LIN {X 0,Y 467.611,Z 154.239,A -85,B 0,C 180,E1 -7725.196,E2 -7725.196} C_VEL
LIN {X 0,Y 467.661,Z 154.233,A -85,B 0,C 180,E1 -7727.854,E2 -7727.854} C_VEL
LIN {X 0,Y 467.686,Z 154.231,A -85,B 0,C 180,E1 -7731.357,E2 -7731.357} C_VEL
LIN {X 0,Y 467.748,Z 154.222,A -85,B 0,C 180,E1 -7733.962,E2 -7733.962} C_VEL
LIN {X 0,Y 467.864,Z 154.208,A -85,B 0,C 180,E1 -7737.417,E2 -7737.417} C_VEL
LIN {X 0,Y 467.888,Z 154.205,A -85,B 0,C 180,E1 -7740,E2 -7740} C_VEL
LIN {X 0,Y 467.863,Z 154.208,A -85,B 0,C 180,E1 -7742.582,E2 -7742.582} C_VEL
LIN {X 0,Y 467.747,Z 154.225,A -85,B 0,C 180,E1 -7746.037,E2 -7746.037} C_VEL
LIN {X 0,Y 467.662,Z 154.235,A -85,B 0,C 180,E1 -7748.643,E2 -7748.643} C_VEL
LIN {X 0,Y 467.382,Z 154.273,A -85,B 0,C 180,E1 -7751.272,E2 -7751.272} C_VEL
LIN {X 0,Y 467.316,Z 155.866,A -85,B 0,C 180,E1 -7753.037,E2 -7753.037} C_VEL
LIN {X 0,Y 467.288,Z 158.633,A -85,B 0,C 180,E1 -7755.727,E2 -7755.727} C_VEL
LIN {X 0,Y 467.15,Z 161.596,A -85,B 0,C 180,E1 -7758.594,E2 -7758.594} C_VEL
LIN {X 0,Y 467.051,Z 165.325,A -85,B 0,C 180,E1 -7762.097,E2 -7762.097} C_VEL
LIN {X 0,Y 467.008,Z 168.875,A -85,B 0,C 180,E1 -7765.452,E2 -7765.452} C_VEL
LIN {X 0,Y 466.965,Z 172.431,A -85,B 0,C 180,E1 -7768.79,E2 -7768.79} C_VEL
LIN {X 0,Y 466.958,Z 173.469,A -85,B 0,C 180,E1 -7769.738,E2 -7769.738} C_VEL
LIN {X 0,Y 470.291,Z 187.316,A -85,B 0,C 180,E1 -7770.288,E2 -7770.288} C_VEL
LIN {X 0,Y 470.011,Z 200.111,A -85,B 0,C 180,E1 -7770.868,E2 -7770.868} C_VEL
LIN {X 0,Y 469.534,Z 212.003,A -85,B 0,C 180,E1 -7771.592,E2 -7771.592} C_VEL
LIN {X 0,Y 469.166,Z 222.158,A -85,B 0,C 180,E1 -7772.379,E2 -7772.379} C_VEL
LIN {X 0,Y 468.706,Z 232.669,A -85,B 0,C 180,E1 -7773.385,E2 -7773.385} C_VEL
LIN {X 0,Y 468.248,Z 242.269,A -85,B 0,C 180,E1 -7774.534,E2 -7774.534} C_VEL
LIN {X 0,Y 467.748,Z 251.276,A -85,B 0,C 180,E1 -7775.872,E2 -7775.872} C_VEL
LIN {X 0,Y 467.449,Z 258.232,A -85,B 0,C 180,E1 -7777.17,E2 -7777.17} C_VEL
LIN {X 0,Y 467.176,Z 264.012,A -85,B 0,C 180,E1 -7778.531,E2 -7778.531} C_VEL
LIN {X 0,Y 466.953,Z 268.413,A -85,B 0,C 180,E1 -7779.862,E2 -7779.862} C_VEL
LIN {X 0,Y 466.786,Z 272.294,A -85,B 0,C 180,E1 -7781.488,E2 -7781.488} C_VEL
LIN {X 0,Y 466.698,Z 274.124,A -85,B 0,C 180,E1 -7782.66,E2 -7782.66} C_VEL
LIN {X 0,Y 466.658,Z 275.233,A -85,B 0,C 180,E1 -7783.849,E2 -7783.849} C_VEL
LIN {X 0,Y 466.63,Z 275.602,A -85,B 0,C 180,E1 -7785.062,E2 -7785.062} C_VEL
LIN {X 0,Y 466.664,Z 275.142,A -85,B 0,C 180,E1 -7786.292,E2 -7786.292} C_VEL
LIN {X 0,Y 466.694,Z 273.843,A -85,B 0,C 180,E1 -7787.552,E2 -7787.552} C_VEL
LIN {X 0,Y 466.803,Z 271.637,A -85,B 0,C 180,E1 -7788.831,E2 -7788.831} C_VEL
LIN {X 0,Y 466.996,Z 267.439,A -85,B 0,C 180,E1 -7790.473,E2 -7790.473} C_VEL
LIN {X 0,Y 467.191,Z 262.264,A -85,B 0,C 180,E1 -7791.919,E2 -7791.919} C_VEL
LIN {X 0,Y 467.459,Z 255.899,A -85,B 0,C 180,E1 -7793.3,E2 -7793.3} C_VEL
LIN {X 0,Y 467.77,Z 249.137,A -85,B 0,C 180,E1 -7794.482,E2 -7794.482} C_VEL
LIN {X 0,Y 468.225,Z 241.035,A -85,B 0,C 180,E1 -7795.643,E2 -7795.643} C_VEL
LIN {X 0,Y 468.607,Z 231.799,A -85,B 0,C 180,E1 -7796.727,E2 -7796.727} C_VEL
LIN {X 0,Y 469.056,Z 221.087,A -85,B 0,C 180,E1 -7797.739,E2 -7797.739} C_VEL
LIN {X 0,Y 469.483,Z 210.135,A -85,B 0,C 180,E1 -7798.568,E2 -7798.568} C_VEL
LIN {X 0,Y 469.942,Z 198.628,A -85,B 0,C 180,E1 -7799.251,E2 -7799.251} C_VEL
LIN {X 0,Y 470.181,Z 187.207,A -85,B 0,C 180,E1 -7799.765,E2 -7799.765} C_VEL
LIN {X 0,Y 467.189,Z 174.165,A -85,B 0,C 180,E1 -7800.28,E2 -7800.28} C_VEL
LIN {X 0,Y 466.844,Z 172.437,A -85,B 0,C 180,E1 -7800.342,E2 -7800.342} C_VEL
LIN {X 0,Y 466.819,Z 171.308,A -85,B 0,C 180,E1 -7801.338,E2 -7801.338} C_VEL
LIN {X 0,Y 466.168,Z 170.562,A -85,B 0,C 180,E1 -7802.053,E2 -7802.053} C_VEL
LIN {X 0,Y 463.366,Z 169.512,A -85,B 0,C 180,E1 -7803.218,E2 -7803.218} C_VEL
LIN {X 0,Y 460.983,Z 168.682,A -85,B 0,C 180,E1 -7804.157,E2 -7804.157} C_VEL
LIN {X 0,Y 459.944,Z 167.972,A -85,B 0,C 180,E1 -7804.881,E2 -7804.881} C_VEL
LIN {X 0,Y 459.852,Z 167.708,A -85,B 0,C 180,E1 -7805.126,E2 -7805.126} C_VEL
LIN {X 0,Y 459.843,Z 164.011,A -85,B 0,C 180,E1 -7808.481,E2 -7808.481} C_VEL
LIN {X 0,Y 459.953,Z 160.915,A -85,B 0,C 180,E1 -7811.323,E2 -7811.323} C_VEL
LIN {X 0,Y 460.058,Z 156.99,A -85,B 0,C 180,E1 -7814.948,E2 -7814.948} C_VEL
LIN {X 0,Y 460.077,Z 155.181,A -85,B 0,C 180,E1 -7816.754,E2 -7816.754} C_VEL
LIN {X 0,Y 460.424,Z 155.134,A -85,B 0,C 180,E1 -7819.445,E2 -7819.445} C_VEL
LIN {X 0,Y 460.681,Z 155.103,A -85,B 0,C 180,E1 -7822.572,E2 -7822.572} C_VEL
LIN {X 0,Y 460.69,Z 155.101,A -85,B 0,C 180,E1 -7824.748,E2 -7824.748} C_VEL
LIN {X 0,Y 460.822,Z 155.083,A -85,B 0,C 180,E1 -7827.377,E2 -7827.377} C_VEL
LIN {X 0,Y 460.85,Z 155.083,A -85,B 0,C 180,E1 -7830,E2 -7830} C_VEL
LIN {X 0,Y 460.822,Z 155.083,A -85,B 0,C 180,E1 -7832.622,E2 -7832.622} C_VEL
LIN {X 0,Y 460.698,Z 155.101,A -85,B 0,C 180,E1 -7836.13,E2 -7836.13} C_VEL
LIN {X 0,Y 460.625,Z 155.107,A -85,B 0,C 180,E1 -7838.776,E2 -7838.776} C_VEL
LIN {X 0,Y 460.61,Z 155.109,A -85,B 0,C 180,E1 -7842.445,E2 -7842.445} C_VEL
LIN {X 0,Y 460.597,Z 155.112,A -85,B 0,C 180,E1 -7845.998,E2 -7845.998} C_VEL
LIN {X 0,Y 460.568,Z 155.114,A -85,B 0,C 180,E1 -7848.902,E2 -7848.902} C_VEL
LIN {X 0,Y 460.513,Z 155.124,A -85,B 0,C 180,E1 -7851.486,E2 -7851.486} C_VEL
LIN {X 0,Y 460.54,Z 155.118,A -85,B 0,C 180,E1 -7854.332,E2 -7854.332} C_VEL
LIN {X 0,Y 460.576,Z 155.115,A -85,B 0,C 180,E1 -7857.244,E2 -7857.244} C_VEL
LIN {X 0,Y 460.508,Z 155.123,A -85,B 0,C 180,E1 -7860.24,E2 -7860.24} C_VEL
LIN {X 0,Y 460.526,Z 155.122,A -85,B 0,C 180,E1 -7863.325,E2 -7863.325} C_VEL
LIN {X 0,Y 460.473,Z 155.128,A -85,B 0,C 180,E1 -7866.53,E2 -7866.53} C_VEL
LIN {X 0,Y 460.53,Z 155.12,A -85,B 0,C 180,E1 -7869.863,E2 -7869.863} C_VEL
LIN {X 0,Y 460.514,Z 155.123,A -85,B 0,C 180,E1 -7872.901,E2 -7872.901} C_VEL
LIN {X 0,Y 460.509,Z 155.123,A -85,B 0,C 180,E1 -7875.831,E2 -7875.831} C_VEL
LIN {X 0,Y 460.529,Z 155.121,A -85,B 0,C 180,E1 -7878.989,E2 -7878.989} C_VEL
LIN {X 0,Y 460.525,Z 155.121,A -85,B 0,C 180,E1 -7881.267,E2 -7881.267} C_VEL
LIN {X 0,Y 460.51,Z 155.125,A -85,B 0,C 180,E1 -7884.555,E2 -7884.555} C_VEL
LIN {X 0,Y 460.529,Z 155.12,A -85,B 0,C 180,E1 -7887.716,E2 -7887.716} C_VEL
LIN {X 0,Y 460.539,Z 155.12,A -85,B 0,C 180,E1 -7890.77,E2 -7890.77} C_VEL
LIN {X 0,Y 460.562,Z 155.116,A -85,B 0,C 180,E1 -7893.735,E2 -7893.735} C_VEL
LIN {X 0,Y 460.545,Z 155.12,A -85,B 0,C 180,E1 -7896.624,E2 -7896.624} C_VEL
LIN {X 0,Y 460.551,Z 155.116,A -85,B 0,C 180,E1 -7899.453,E2 -7899.453} C_VEL
LIN {X 0,Y 460.549,Z 155.119,A -85,B 0,C 180,E1 -7902.23,E2 -7902.23} C_VEL
LIN {X 0,Y 460.565,Z 155.115,A -85,B 0,C 180,E1 -7904.965,E2 -7904.965} C_VEL
LIN {X 0,Y 460.612,Z 155.111,A -85,B 0,C 180,E1 -7908.56,E2 -7908.56} C_VEL
LIN {X 0,Y 460.666,Z 155.106,A -85,B 0,C 180,E1 -7912.109,E2 -7912.109} C_VEL
LIN {X 0,Y 460.698,Z 155.099,A -85,B 0,C 180,E1 -7914.749,E2 -7914.749} C_VEL
LIN {X 0,Y 460.826,Z 155.083,A -85,B 0,C 180,E1 -7917.378,E2 -7917.378} C_VEL
LIN {X 0,Y 460.855,Z 155.081,A -85,B 0,C 180,E1 -7920,E2 -7920} C_VEL
LIN {X 0,Y 460.802,Z 155.087,A -85,B 0,C 180,E1 -7922.623,E2 -7922.623} C_VEL
LIN {X 0,Y 460.689,Z 155.102,A -85,B 0,C 180,E1 -7926.131,E2 -7926.131} C_VEL
LIN {X 0,Y 460.621,Z 155.109,A -85,B 0,C 180,E1 -7928.777,E2 -7928.777} C_VEL
LIN {X 0,Y 460.616,Z 155.11,A -85,B 0,C 180,E1 -7932.445,E2 -7932.445} C_VEL
LIN {X 0,Y 460.602,Z 155.113,A -85,B 0,C 180,E1 -7935.998,E2 -7935.998} C_VEL
LIN {X 0,Y 460.573,Z 155.115,A -85,B 0,C 180,E1 -7938.902,E2 -7938.902} C_VEL
LIN {X 0,Y 460.518,Z 155.123,A -85,B 0,C 180,E1 -7941.486,E2 -7941.486} C_VEL
LIN {X 0,Y 460.544,Z 155.118,A -85,B 0,C 180,E1 -7944.333,E2 -7944.333} C_VEL
LIN {X 0,Y 460.576,Z 155.117,A -85,B 0,C 180,E1 -7947.244,E2 -7947.244} C_VEL
LIN {X 0,Y 460.513,Z 155.122,A -85,B 0,C 180,E1 -7950.24,E2 -7950.24} C_VEL
LIN {X 0,Y 460.522,Z 155.123,A -85,B 0,C 180,E1 -7953.326,E2 -7953.326} C_VEL
LIN {X 0,Y 460.478,Z 155.126,A -85,B 0,C 180,E1 -7956.53,E2 -7956.53} C_VEL
LIN {X 0,Y 460.529,Z 155.12,A -85,B 0,C 180,E1 -7959.863,E2 -7959.863} C_VEL
LIN {X 0,Y 460.516,Z 155.12,A -85,B 0,C 180,E1 -7962.901,E2 -7962.901} C_VEL
LIN {X 0,Y 460.512,Z 155.119,A -85,B 0,C 180,E1 -7965.831,E2 -7965.831} C_VEL
LIN {X 0,Y 460.568,Z 155.274,A -85,B 0,C 180,E1 -7968.772,E2 -7968.772} C_VEL
LIN {X 0,Y 461.803,Z 162.028,A -85,B 0,C 180,E1 -7971.886,E2 -7971.886} C_VEL
LIN {X 0,Y 462.375,Z 166.113,A -85,B 0,C 180,E1 -7973.668,E2 -7973.668} C_VEL
LIN {X 0,Y 462.315,Z 169.762,A -85,B 0,C 180,E1 -7975.175,E2 -7975.175} C_VEL
LIN {X 0,Y 461.89,Z 178.017,A -85,B 0,C 180,E1 -7978.439,E2 -7978.439} C_VEL
LIN {X 0,Y 461.411,Z 186.948,A -85,B 0,C 180,E1 -7981.824,E2 -7981.824} C_VEL
LIN {X 0,Y 461.022,Z 194.814,A -85,B 0,C 180,E1 -7984.733,E2 -7984.733} C_VEL
LIN {X 0,Y 460.698,Z 204.34,A -85,B 0,C 180,E1 -7988.053,E2 -7988.053} C_VEL
LIN {X 0,Y 460.425,Z 213.922,A -85,B 0,C 180,E1 -7991.304,E2 -7991.304} C_VEL
LIN {X 0,Y 460.171,Z 223.123,A -85,B 0,C 180,E1 -7994.353,E2 -7994.353} C_VEL
LIN {X 0,Y 462.462,Z 236.69,A -85,B 0,C 180,E1 -7994.786,E2 -7994.786} C_VEL
LIN {X 0,Y 463.251,Z 243.184,A -85,B 0,C 180,E1 -7995.054,E2 -7995.054} C_VEL
LIN {X 0,Y 462.828,Z 254.843,A -85,B 0,C 180,E1 -7995.602,E2 -7995.602} C_VEL
LIN {X 0,Y 462.299,Z 267.178,A -85,B 0,C 180,E1 -7996.371,E2 -7996.371} C_VEL
LIN {X 0,Y 461.847,Z 277.169,A -85,B 0,C 180,E1 -7997.161,E2 -7997.161} C_VEL
LIN {X 0,Y 461.404,Z 287.178,A -85,B 0,C 180,E1 -7998.134,E2 -7998.134} C_VEL
LIN {X 0,Y 460.86,Z 296.393,A -85,B 0,C 180,E1 -7999.233,E2 -7999.233} C_VEL
LIN {X 0,Y 460.418,Z 305.381,A -85,B 0,C 180,E1 -8000.556,E2 -8000.556} C_VEL
LIN {X 0,Y 460.055,Z 312.619,A -85,B 0,C 180,E1 -8001.877,E2 -8001.877} C_VEL
LIN {X 0,Y 459.848,Z 317.508,A -85,B 0,C 180,E1 -8002.977,E2 -8002.977} C_VEL
LIN {X 0,Y 459.754,Z 322.266,A -85,B 0,C 180,E1 -8004.298,E2 -8004.298} C_VEL
LIN {X 0,Y 459.58,Z 325.896,A -85,B 0,C 180,E1 -8005.615,E2 -8005.615} C_VEL
LIN {X 0,Y 459.591,Z 327.773,A -85,B 0,C 180,E1 -8006.493,E2 -8006.493} C_VEL
LIN {X 0,Y 459.571,Z 329.175,A -85,B 0,C 180,E1 -8007.371,E2 -8007.371} C_VEL
LIN {X 0,Y 459.495,Z 330.779,A -85,B 0,C 180,E1 -8009.124,E2 -8009.124} C_VEL
LIN {X 0,Y 459.474,Z 330.994,A -85,B 0,C 180,E1 -8010,E2 -8010} C_VEL
LIN {X 0,Y 459.495,Z 330.779,A -85,B 0,C 180,E1 -8010.877,E2 -8010.877} C_VEL
LIN {X 0,Y 459.571,Z 329.178,A -85,B 0,C 180,E1 -8012.63,E2 -8012.63} C_VEL
LIN {X 0,Y 459.591,Z 327.777,A -85,B 0,C 180,E1 -8013.507,E2 -8013.507} C_VEL
LIN {X 0,Y 459.635,Z 324.817,A -85,B 0,C 180,E1 -8014.824,E2 -8014.824} C_VEL
LIN {X 0,Y 459.758,Z 320.814,A -85,B 0,C 180,E1 -8016.143,E2 -8016.143} C_VEL
LIN {X 0,Y 459.93,Z 314.654,A -85,B 0,C 180,E1 -8017.684,E2 -8017.684} C_VEL
LIN {X 0,Y 460.288,Z 307.933,A -85,B 0,C 180,E1 -8019.004,E2 -8019.004} C_VEL
LIN {X 0,Y 460.702,Z 299.594,A -85,B 0,C 180,E1 -8020.326,E2 -8020.326} C_VEL
LIN {X 0,Y 461.133,Z 291.05,A -85,B 0,C 180,E1 -8021.428,E2 -8021.428} C_VEL
LIN {X 0,Y 461.671,Z 280.881,A -85,B 0,C 180,E1 -8022.493,E2 -8022.493} C_VEL
LIN {X 0,Y 462.114,Z 270.071,A -85,B 0,C 180,E1 -8023.411,E2 -8023.411} C_VEL
LIN {X 0,Y 462.639,Z 258.657,A -85,B 0,C 180,E1 -8024.179,E2 -8024.179} C_VEL
LIN {X 0,Y 463.138,Z 246.96,A -85,B 0,C 180,E1 -8024.781,E2 -8024.781} C_VEL
LIN {X 0,Y 463.081,Z 240.887,A -85,B 0,C 180,E1 -8025.036,E2 -8025.036} C_VEL
LIN {X 0,Y 460.877,Z 227.519,A -85,B 0,C 180,E1 -8025.524,E2 -8025.524} C_VEL
LIN {X 0,Y 460.147,Z 222.604,A -85,B 0,C 180,E1 -8025.689,E2 -8025.689} C_VEL
LIN {X 0,Y 460.455,Z 212.219,A -85,B 0,C 180,E1 -8029.179,E2 -8029.179} C_VEL
LIN {X 0,Y 460.708,Z 202.589,A -85,B 0,C 180,E1 -8032.419,E2 -8032.419} C_VEL
LIN {X 0,Y 460.989,Z 194.447,A -85,B 0,C 180,E1 -8035.27,E2 -8035.27} C_VEL
LIN {X 0,Y 461.354,Z 186.345,A -85,B 0,C 180,E1 -8038.18,E2 -8038.18} C_VEL
LIN {X 0,Y 461.761,Z 177.524,A -85,B 0,C 180,E1 -8041.534,E2 -8041.534} C_VEL
LIN {X 0,Y 462.195,Z 170.722,A -85,B 0,C 180,E1 -8044.237,E2 -8044.237} C_VEL
LIN {X 0,Y 462.427,Z 166.976,A -85,B 0,C 180,E1 -8045.797,E2 -8045.797} C_VEL
LIN {X 0,Y 461.926,Z 162.705,A -85,B 0,C 180,E1 -8047.706,E2 -8047.706} C_VEL
LIN {X 0,Y 460.705,Z 155.996,A -85,B 0,C 180,E1 -8050.993,E2 -8050.993} C_VEL
LIN {X 0,Y 460.53,Z 155.123,A -85,B 0,C 180,E1 -8051.493,E2 -8051.493} C_VEL
LIN {X 0,Y 460.521,Z 155.123,A -85,B 0,C 180,E1 -8054.588,E2 -8054.588} C_VEL
LIN {X 0,Y 460.527,Z 155.125,A -85,B 0,C 180,E1 -8057.819,E2 -8057.819} C_VEL
LIN {X 0,Y 460.549,Z 155.121,A -85,B 0,C 180,E1 -8061.102,E2 -8061.102} C_VEL
LIN {X 0,Y 460.515,Z 155.125,A -85,B 0,C 180,E1 -8064.554,E2 -8064.554} C_VEL
LIN {X 0,Y 460.536,Z 155.121,A -85,B 0,C 180,E1 -8067.716,E2 -8067.716} C_VEL
LIN {X 0,Y 460.545,Z 155.119,A -85,B 0,C 180,E1 -8070.769,E2 -8070.769} C_VEL
LIN {X 0,Y 460.568,Z 155.117,A -85,B 0,C 180,E1 -8073.735,E2 -8073.735} C_VEL
LIN {X 0,Y 460.551,Z 155.119,A -85,B 0,C 180,E1 -8076.624,E2 -8076.624} C_VEL
LIN {X 0,Y 460.556,Z 155.117,A -85,B 0,C 180,E1 -8079.453,E2 -8079.453} C_VEL
LIN {X 0,Y 460.554,Z 155.116,A -85,B 0,C 180,E1 -8082.23,E2 -8082.23} C_VEL
LIN {X 0,Y 460.57,Z 155.116,A -85,B 0,C 180,E1 -8084.965,E2 -8084.965} C_VEL
LIN {X 0,Y 460.616,Z 155.112,A -85,B 0,C 180,E1 -8088.559,E2 -8088.559} C_VEL
LIN {X 0,Y 460.7,Z 155.1,A -85,B 0,C 180,E1 -8092.108,E2 -8092.108} C_VEL
LIN {X 0,Y 460.702,Z 155.101,A -85,B 0,C 180,E1 -8094.748,E2 -8094.748} C_VEL
LIN {X 0,Y 460.829,Z 155.084,A -85,B 0,C 180,E1 -8097.377,E2 -8097.377} C_VEL
LIN {X 0,Y 460.858,Z 155.081,A -85,B 0,C 180,E1 -8100,E2 -8100} C_VEL
LIN {X 0,Y 460.828,Z 155.085,A -85,B 0,C 180,E1 -8102.622,E2 -8102.622} C_VEL
LIN {X 0,Y 460.713,Z 155.101,A -85,B 0,C 180,E1 -8106.129,E2 -8106.129} C_VEL
LIN {X 0,Y 460.602,Z 155.114,A -85,B 0,C 180,E1 -8108.776,E2 -8108.776} C_VEL
LIN {X 0,Y 460.338,Z 155.15,A -85,B 0,C 180,E1 -8111.447,E2 -8111.447} C_VEL
LIN {X 0,Y 460.24,Z 157.881,A -85,B 0,C 180,E1 -8114.141,E2 -8114.141} C_VEL
LIN {X 0,Y 460.151,Z 160.654,A -85,B 0,C 180,E1 -8116.869,E2 -8116.869} C_VEL
LIN {X 0,Y 460.026,Z 163.534,A -85,B 0,C 180,E1 -8119.639,E2 -8119.639} C_VEL
LIN {X 0,Y 460.006,Z 166.49,A -85,B 0,C 180,E1 -8122.454,E2 -8122.454} C_VEL
LIN {X 0,Y 459.936,Z 169.824,A -85,B 0,C 180,E1 -8125.638,E2 -8125.638} C_VEL
LIN {X 0,Y 459.895,Z 172.627,A -85,B 0,C 180,E1 -8128.276,E2 -8128.276} C_VEL
LIN {X 0,Y 459.907,Z 173.921,A -85,B 0,C 180,E1 -8129.485,E2 -8129.485} C_VEL
LIN {X 0,Y 463.241,Z 187.446,A -85,B 0,C 180,E1 -8130.043,E2 -8130.043} C_VEL
LIN {X 0,Y 463.479,Z 190.923,A -85,B 0,C 180,E1 -8130.194,E2 -8130.194} C_VEL
LIN {X 0,Y 463.083,Z 202.927,A -85,B 0,C 180,E1 -8130.785,E2 -8130.785} C_VEL
LIN {X 0,Y 462.612,Z 214.1,A -85,B 0,C 180,E1 -8131.505,E2 -8131.505} C_VEL
LIN {X 0,Y 462.154,Z 225.169,A -85,B 0,C 180,E1 -8132.414,E2 -8132.414} C_VEL
LIN {X 0,Y 461.658,Z 235.629,A -85,B 0,C 180,E1 -8133.493,E2 -8133.493} C_VEL
LIN {X 0,Y 461.181,Z 244.529,A -85,B 0,C 180,E1 -8134.622,E2 -8134.622} C_VEL
LIN {X 0,Y 460.748,Z 251.676,A -85,B 0,C 180,E1 -8135.724,E2 -8135.724} C_VEL
LIN {X 0,Y 460.421,Z 258.398,A -85,B 0,C 180,E1 -8136.988,E2 -8136.988} C_VEL
LIN {X 0,Y 460.126,Z 264.679,A -85,B 0,C 180,E1 -8138.492,E2 -8138.492} C_VEL
LIN {X 0,Y 459.881,Z 269.267,A -85,B 0,C 180,E1 -8139.929,E2 -8139.929} C_VEL
LIN {X 0,Y 459.715,Z 272.844,A -85,B 0,C 180,E1 -8141.487,E2 -8141.487} C_VEL
LIN {X 0,Y 459.61,Z 274.756,A -85,B 0,C 180,E1 -8142.779,E2 -8142.779} C_VEL
LIN {X 0,Y 459.557,Z 275.781,A -85,B 0,C 180,E1 -8144.047,E2 -8144.047} C_VEL
LIN {X 0,Y 459.538,Z 275.988,A -85,B 0,C 180,E1 -8145.291,E2 -8145.291} C_VEL
LIN {X 0,Y 459.581,Z 275.427,A -85,B 0,C 180,E1 -8146.516,E2 -8146.516} C_VEL
LIN {X 0,Y 459.631,Z 274.094,A -85,B 0,C 180,E1 -8147.717,E2 -8147.717} C_VEL
LIN {X 0,Y 459.726,Z 272.024,A -85,B 0,C 180,E1 -8148.901,E2 -8148.901} C_VEL
LIN {X 0,Y 459.857,Z 269.234,A -85,B 0,C 180,E1 -8150.067,E2 -8150.067} C_VEL
LIN {X 0,Y 460.064,Z 264.654,A -85,B 0,C 180,E1 -8151.501,E2 -8151.501} C_VEL
LIN {X 0,Y 460.346,Z 258.317,A -85,B 0,C 180,E1 -8153.016,E2 -8153.016} C_VEL
LIN {X 0,Y 460.656,Z 251.668,A -85,B 0,C 180,E1 -8154.273,E2 -8154.273} C_VEL
LIN {X 0,Y 461.11,Z 243.866,A -85,B 0,C 180,E1 -8155.468,E2 -8155.468} C_VEL
LIN {X 0,Y 461.569,Z 234.591,A -85,B 0,C 180,E1 -8156.629,E2 -8156.629} C_VEL
LIN {X 0,Y 462.04,Z 223.998,A -85,B 0,C 180,E1 -8157.705,E2 -8157.705} C_VEL
LIN {X 0,Y 462.468,Z 212.881,A -85,B 0,C 180,E1 -8158.601,E2 -8158.601} C_VEL
LIN {X 0,Y 462.995,Z 201.026,A -85,B 0,C 180,E1 -8159.347,E2 -8159.347} C_VEL
LIN {X 0,Y 463.371,Z 189.539,A -85,B 0,C 180,E1 -8159.898,E2 -8159.898} C_VEL
LIN {X 0,Y 461.195,Z 178.757,A -85,B 0,C 180,E1 -8160.36,E2 -8160.36} C_VEL
LIN {X 0,Y 459.774,Z 172.801,A -85,B 0,C 180,E1 -8160.589,E2 -8160.589} C_VEL
LIN {X 0,Y 459.831,Z 169.306,A -85,B 0,C 180,E1 -8163.689,E2 -8163.689} C_VEL
LIN {X 0,Y 459.852,Z 167.708,A -85,B 0,C 180,E1 -8165.126,E2 -8165.126} C_VEL
LIN {X 0,Y 459.155,Z 166.978,A -85,B 0,C 180,E1 -8165.851,E2 -8165.851} C_VEL
LIN {X 0,Y 456.273,Z 165.947,A -85,B 0,C 180,E1 -8167.03,E2 -8167.03} C_VEL
LIN {X 0,Y 453.866,Z 165.145,A -85,B 0,C 180,E1 -8167.982,E2 -8167.982} C_VEL
LIN {X 0,Y 452.857,Z 164.451,A -85,B 0,C 180,E1 -8168.717,E2 -8168.717} C_VEL
LIN {X 0,Y 452.786,Z 164.187,A -85,B 0,C 180,E1 -8168.965,E2 -8168.965} C_VEL
LIN {X 0,Y 452.894,Z 160.989,A -85,B 0,C 180,E1 -8171.919,E2 -8171.919} C_VEL
LIN {X 0,Y 452.999,Z 157.975,A -85,B 0,C 180,E1 -8174.707,E2 -8174.707} C_VEL
LIN {X 0,Y 452.994,Z 156.068,A -85,B 0,C 180,E1 -8176.543,E2 -8176.543} C_VEL
LIN {X 0,Y 453.36,Z 156.013,A -85,B 0,C 180,E1 -8179.279,E2 -8179.279} C_VEL
LIN {X 0,Y 453.6,Z 155.985,A -85,B 0,C 180,E1 -8181.984,E2 -8181.984} C_VEL
LIN {X 0,Y 453.663,Z 155.976,A -85,B 0,C 180,E1 -8184.666,E2 -8184.666} C_VEL
LIN {X 0,Y 453.762,Z 155.962,A -85,B 0,C 180,E1 -8187.337,E2 -8187.337} C_VEL
LIN {X 0,Y 453.821,Z 155.959,A -85,B 0,C 180,E1 -8190,E2 -8190} C_VEL
LIN {X 0,Y 453.762,Z 155.962,A -85,B 0,C 180,E1 -8192.663,E2 -8192.663} C_VEL
LIN {X 0,Y 453.665,Z 155.976,A -85,B 0,C 180,E1 -8196.225,E2 -8196.225} C_VEL
LIN {X 0,Y 453.589,Z 155.984,A -85,B 0,C 180,E1 -8198.913,E2 -8198.913} C_VEL
LIN {X 0,Y 453.56,Z 155.987,A -85,B 0,C 180,E1 -8202.529,E2 -8202.529} C_VEL
LIN {X 0,Y 453.541,Z 155.991,A -85,B 0,C 180,E1 -8206.196,E2 -8206.196} C_VEL
LIN {X 0,Y 453.517,Z 155.993,A -85,B 0,C 180,E1 -8209.041,E2 -8209.041} C_VEL
LIN {X 0,Y 453.473,Z 156,A -85,B 0,C 180,E1 -8211.836,E2 -8211.836} C_VEL
LIN {X 0,Y 453.511,Z 155.994,A -85,B 0,C 180,E1 -8214.735,E2 -8214.735} C_VEL
LIN {X 0,Y 453.534,Z 155.991,A -85,B 0,C 180,E1 -8217.961,E2 -8217.961} C_VEL
LIN {X 0,Y 453.463,Z 156.002,A -85,B 0,C 180,E1 -8221.525,E2 -8221.525} C_VEL
LIN {X 0,Y 453.484,Z 155.998,A -85,B 0,C 180,E1 -8224.778,E2 -8224.778} C_VEL
LIN {X 0,Y 453.462,Z 156,A -85,B 0,C 180,E1 -8228.312,E2 -8228.312} C_VEL
LIN {X 0,Y 453.491,Z 155.997,A -85,B 0,C 180,E1 -8230.609,E2 -8230.609} C_VEL
LIN {X 0,Y 453.47,Z 155.998,A -85,B 0,C 180,E1 -8234.221,E2 -8234.221} C_VEL
LIN {X 0,Y 453.461,Z 156.003,A -85,B 0,C 180,E1 -8237.006,E2 -8237.006} C_VEL
LIN {X 0,Y 453.503,Z 155.996,A -85,B 0,C 180,E1 -8240.552,E2 -8240.552} C_VEL
LIN {X 0,Y 453.454,Z 156,A -85,B 0,C 180,E1 -8243.918,E2 -8243.918} C_VEL
LIN {X 0,Y 453.48,Z 155.999,A -85,B 0,C 180,E1 -8247.152,E2 -8247.152} C_VEL
LIN {X 0,Y 453.473,Z 156,A -85,B 0,C 180,E1 -8250.269,E2 -8250.269} C_VEL
LIN {X 0,Y 453.506,Z 155.995,A -85,B 0,C 180,E1 -8253.294,E2 -8253.294} C_VEL
LIN {X 0,Y 453.502,Z 155.996,A -85,B 0,C 180,E1 -8256.239,E2 -8256.239} C_VEL
LIN {X 0,Y 453.482,Z 155.997,A -85,B 0,C 180,E1 -8259.118,E2 -8259.118} C_VEL
LIN {X 0,Y 453.504,Z 155.995,A -85,B 0,C 180,E1 -8261.945,E2 -8261.945} C_VEL
LIN {X 0,Y 453.54,Z 155.993,A -85,B 0,C 180,E1 -8264.727,E2 -8264.727} C_VEL
LIN {X 0,Y 453.561,Z 155.991,A -85,B 0,C 180,E1 -8268.379,E2 -8268.379} C_VEL
LIN {X 0,Y 453.587,Z 155.984,A -85,B 0,C 180,E1 -8271.087,E2 -8271.087} C_VEL
LIN {X 0,Y 453.674,Z 155.975,A -85,B 0,C 180,E1 -8273.775,E2 -8273.775} C_VEL
LIN {X 0,Y 453.767,Z 155.962,A -85,B 0,C 180,E1 -8277.337,E2 -8277.337} C_VEL
LIN {X 0,Y 453.825,Z 155.956,A -85,B 0,C 180,E1 -8280,E2 -8280} C_VEL
LIN {X 0,Y 453.746,Z 155.966,A -85,B 0,C 180,E1 -8282.664,E2 -8282.664} C_VEL
LIN {X 0,Y 453.655,Z 155.978,A -85,B 0,C 180,E1 -8286.226,E2 -8286.226} C_VEL
LIN {X 0,Y 453.587,Z 155.985,A -85,B 0,C 180,E1 -8288.914,E2 -8288.914} C_VEL
LIN {X 0,Y 453.566,Z 155.988,A -85,B 0,C 180,E1 -8292.529,E2 -8292.529} C_VEL
LIN {X 0,Y 453.547,Z 155.991,A -85,B 0,C 180,E1 -8296.196,E2 -8296.196} C_VEL
LIN {X 0,Y 453.523,Z 155.994,A -85,B 0,C 180,E1 -8299.041,E2 -8299.041} C_VEL
LIN {X 0,Y 453.479,Z 156,A -85,B 0,C 180,E1 -8301.836,E2 -8301.836} C_VEL
LIN {X 0,Y 453.516,Z 155.994,A -85,B 0,C 180,E1 -8304.735,E2 -8304.735} C_VEL
LIN {X 0,Y 453.535,Z 155.993,A -85,B 0,C 180,E1 -8307.96,E2 -8307.96} C_VEL
LIN {X 0,Y 453.468,Z 156.001,A -85,B 0,C 180,E1 -8311.525,E2 -8311.525} C_VEL
LIN {X 0,Y 453.484,Z 155.999,A -85,B 0,C 180,E1 -8314.777,E2 -8314.777} C_VEL
LIN {X 0,Y 453.465,Z 156,A -85,B 0,C 180,E1 -8318.312,E2 -8318.312} C_VEL
LIN {X 0,Y 453.496,Z 155.998,A -85,B 0,C 180,E1 -8320.609,E2 -8320.609} C_VEL
LIN {X 0,Y 453.458,Z 155.998,A -85,B 0,C 180,E1 -8323.244,E2 -8323.244} C_VEL
LIN {X 0,Y 453.467,Z 155.996,A -85,B 0,C 180,E1 -8325.779,E2 -8325.779} C_VEL
LIN {X 0,Y 453.521,Z 156.126,A -85,B 0,C 180,E1 -8328.437,E2 -8328.437} C_VEL
LIN {X 0,Y 454.64,Z 162.079,A -85,B 0,C 180,E1 -8331.247,E2 -8331.247} C_VEL
LIN {X 0,Y 455.348,Z 166.819,A -85,B 0,C 180,E1 -8333.378,E2 -8333.378} C_VEL
LIN {X 0,Y 455.323,Z 171.095,A -85,B 0,C 180,E1 -8335.173,E2 -8335.173} C_VEL
LIN {X 0,Y 454.91,Z 178.895,A -85,B 0,C 180,E1 -8338.313,E2 -8338.313} C_VEL
LIN {X 0,Y 454.434,Z 186.775,A -85,B 0,C 180,E1 -8341.352,E2 -8341.352} C_VEL
LIN {X 0,Y 454.043,Z 194.642,A -85,B 0,C 180,E1 -8344.316,E2 -8344.316} C_VEL
LIN {X 0,Y 453.718,Z 202.695,A -85,B 0,C 180,E1 -8347.217,E2 -8347.217} C_VEL
LIN {X 0,Y 453.458,Z 210.923,A -85,B 0,C 180,E1 -8350.064,E2 -8350.064} C_VEL
LIN {X 0,Y 453.157,Z 220.336,A -85,B 0,C 180,E1 -8353.327,E2 -8353.327} C_VEL
LIN {X 0,Y 453.079,Z 222.553,A -85,B 0,C 180,E1 -8354.097,E2 -8354.097} C_VEL
LIN {X 0,Y 455.342,Z 235.998,A -85,B 0,C 180,E1 -8354.533,E2 -8354.533} C_VEL
LIN {X 0,Y 456.342,Z 244.086,A -85,B 0,C 180,E1 -8354.88,E2 -8354.88} C_VEL
LIN {X 0,Y 455.823,Z 256.42,A -85,B 0,C 180,E1 -8355.49,E2 -8355.49} C_VEL
LIN {X 0,Y 455.293,Z 268.304,A -85,B 0,C 180,E1 -8356.271,E2 -8356.271} C_VEL
LIN {X 0,Y 454.778,Z 278.84,A -85,B 0,C 180,E1 -8357.152,E2 -8357.152} C_VEL
LIN {X 0,Y 454.291,Z 288.725,A -85,B 0,C 180,E1 -8358.172,E2 -8358.172} C_VEL
LIN {X 0,Y 453.726,Z 297.613,A -85,B 0,C 180,E1 -8359.288,E2 -8359.288} C_VEL
LIN {X 0,Y 453.31,Z 306.295,A -85,B 0,C 180,E1 -8360.631,E2 -8360.631} C_VEL
LIN {X 0,Y 452.925,Z 313.234,A -85,B 0,C 180,E1 -8361.972,E2 -8361.972} C_VEL
LIN {X 0,Y 452.731,Z 319.374,A -85,B 0,C 180,E1 -8363.471,E2 -8363.471} C_VEL
LIN {X 0,Y 452.567,Z 324.405,A -85,B 0,C 180,E1 -8365.101,E2 -8365.101} C_VEL
LIN {X 0,Y 452.493,Z 327.359,A -85,B 0,C 180,E1 -8366.438,E2 -8366.438} C_VEL
LIN {X 0,Y 452.496,Z 328.767,A -85,B 0,C 180,E1 -8367.329,E2 -8367.329} C_VEL
LIN {X 0,Y 452.433,Z 330.381,A -85,B 0,C 180,E1 -8369.11,E2 -8369.11} C_VEL
LIN {X 0,Y 452.411,Z 330.596,A -85,B 0,C 180,E1 -8370,E2 -8370} C_VEL
LIN {X 0,Y 452.433,Z 330.378,A -85,B 0,C 180,E1 -8370.89,E2 -8370.89} C_VEL
LIN {X 0,Y 452.496,Z 328.761,A -85,B 0,C 180,E1 -8372.671,E2 -8372.671} C_VEL
LIN {X 0,Y 452.494,Z 327.348,A -85,B 0,C 180,E1 -8373.562,E2 -8373.562} C_VEL
LIN {X 0,Y 452.567,Z 324.385,A -85,B 0,C 180,E1 -8374.9,E2 -8374.9} C_VEL
LIN {X 0,Y 452.692,Z 319.499,A -85,B 0,C 180,E1 -8376.486,E2 -8376.486} C_VEL
LIN {X 0,Y 452.927,Z 313.189,A -85,B 0,C 180,E1 -8378.028,E2 -8378.028} C_VEL
LIN {X 0,Y 453.3,Z 306.232,A -85,B 0,C 180,E1 -8379.369,E2 -8379.369} C_VEL
LIN {X 0,Y 453.712,Z 297.529,A -85,B 0,C 180,E1 -8380.713,E2 -8380.713} C_VEL
LIN {X 0,Y 454.282,Z 288.622,A -85,B 0,C 180,E1 -8381.829,E2 -8381.829} C_VEL
LIN {X 0,Y 454.788,Z 278.801,A -85,B 0,C 180,E1 -8382.839,E2 -8382.839} C_VEL
LIN {X 0,Y 455.249,Z 268.16,A -85,B 0,C 180,E1 -8383.731,E2 -8383.731} C_VEL
LIN {X 0,Y 455.823,Z 256.242,A -85,B 0,C 180,E1 -8384.51,E2 -8384.51} C_VEL
LIN {X 0,Y 456.338,Z 243.875,A -85,B 0,C 180,E1 -8385.121,E2 -8385.121} C_VEL
LIN {X 0,Y 454.579,Z 231.503,A -85,B 0,C 180,E1 -8385.628,E2 -8385.628} C_VEL
LIN {X 0,Y 453.079,Z 222.268,A -85,B 0,C 180,E1 -8385.903,E2 -8385.903} C_VEL
LIN {X 0,Y 453.41,Z 211.85,A -85,B 0,C 180,E1 -8389.467,E2 -8389.467} C_VEL
LIN {X 0,Y 453.682,Z 202.231,A -85,B 0,C 180,E1 -8392.785,E2 -8392.785} C_VEL
LIN {X 0,Y 454.04,Z 192.856,A -85,B 0,C 180,E1 -8396.133,E2 -8396.133} C_VEL
LIN {X 0,Y 454.412,Z 184.789,A -85,B 0,C 180,E1 -8399.156,E2 -8399.156} C_VEL
LIN {X 0,Y 454.882,Z 176.973,A -85,B 0,C 180,E1 -8402.214,E2 -8402.214} C_VEL
LIN {X 0,Y 455.381,Z 169.895,A -85,B 0,C 180,E1 -8405.118,E2 -8405.118} C_VEL
LIN {X 0,Y 455.248,Z 165.605,A -85,B 0,C 180,E1 -8407.019,E2 -8407.019} C_VEL
LIN {X 0,Y 453.909,Z 158.194,A -85,B 0,C 180,E1 -8410.651,E2 -8410.651} C_VEL
LIN {X 0,Y 453.48,Z 156,A -85,B 0,C 180,E1 -8411.935,E2 -8411.935} C_VEL
LIN {X 0,Y 453.492,Z 156,A -85,B 0,C 180,E1 -8415.471,E2 -8415.471} C_VEL
LIN {X 0,Y 453.483,Z 156.002,A -85,B 0,C 180,E1 -8418.209,E2 -8418.209} C_VEL
LIN {X 0,Y 453.52,Z 155.996,A -85,B 0,C 180,E1 -8420.79,E2 -8420.79} C_VEL
LIN {X 0,Y 453.459,Z 156.002,A -85,B 0,C 180,E1 -8423.917,E2 -8423.917} C_VEL
LIN {X 0,Y 453.487,Z 155.999,A -85,B 0,C 180,E1 -8427.151,E2 -8427.151} C_VEL
LIN {X 0,Y 453.48,Z 156.001,A -85,B 0,C 180,E1 -8430.268,E2 -8430.268} C_VEL
LIN {X 0,Y 453.514,Z 155.994,A -85,B 0,C 180,E1 -8433.294,E2 -8433.294} C_VEL
LIN {X 0,Y 453.508,Z 155.997,A -85,B 0,C 180,E1 -8436.239,E2 -8436.239} C_VEL
LIN {X 0,Y 453.487,Z 155.999,A -85,B 0,C 180,E1 -8439.117,E2 -8439.117} C_VEL
LIN {X 0,Y 453.508,Z 155.993,A -85,B 0,C 180,E1 -8441.944,E2 -8441.944} C_VEL
LIN {X 0,Y 453.544,Z 155.991,A -85,B 0,C 180,E1 -8444.726,E2 -8444.726} C_VEL
LIN {X 0,Y 453.565,Z 155.99,A -85,B 0,C 180,E1 -8448.379,E2 -8448.379} C_VEL
LIN {X 0,Y 453.657,Z 155.977,A -85,B 0,C 180,E1 -8451.985,E2 -8451.985} C_VEL
LIN {X 0,Y 453.676,Z 155.977,A -85,B 0,C 180,E1 -8454.666,E2 -8454.666} C_VEL
LIN {X 0,Y 453.769,Z 155.964,A -85,B 0,C 180,E1 -8457.336,E2 -8457.336} C_VEL
LIN {X 0,Y 453.829,Z 155.957,A -85,B 0,C 180,E1 -8460,E2 -8460} C_VEL
LIN {X 0,Y 453.768,Z 155.964,A -85,B 0,C 180,E1 -8462.663,E2 -8462.663} C_VEL
LIN {X 0,Y 453.681,Z 155.977,A -85,B 0,C 180,E1 -8466.225,E2 -8466.225} C_VEL
LIN {X 0,Y 453.559,Z 155.991,A -85,B 0,C 180,E1 -8468.914,E2 -8468.914} C_VEL
LIN {X 0,Y 453.299,Z 156.23,A -85,B 0,C 180,E1 -8471.627,E2 -8471.627} C_VEL
LIN {X 0,Y 453.199,Z 158.973,A -85,B 0,C 180,E1 -8474.366,E2 -8474.366} C_VEL
LIN {X 0,Y 453.084,Z 161.772,A -85,B 0,C 180,E1 -8477.14,E2 -8477.14} C_VEL
LIN {X 0,Y 452.976,Z 164.707,A -85,B 0,C 180,E1 -8479.958,E2 -8479.958} C_VEL
LIN {X 0,Y 452.915,Z 167.668,A -85,B 0,C 180,E1 -8482.825,E2 -8482.825} C_VEL
LIN {X 0,Y 452.862,Z 170.787,A -85,B 0,C 180,E1 -8485.827,E2 -8485.827} C_VEL
LIN {X 0,Y 452.822,Z 174.149,A -85,B 0,C 180,E1 -8489.013,E2 -8489.013} C_VEL
LIN {X 0,Y 452.839,Z 174.388,A -85,B 0,C 180,E1 -8489.234,E2 -8489.234} C_VEL
LIN {X 0,Y 456.488,Z 189.117,A -85,B 0,C 180,E1 -8489.86,E2 -8489.86} C_VEL
LIN {X 0,Y 456.35,Z 200.655,A -85,B 0,C 180,E1 -8490.409,E2 -8490.409} C_VEL
LIN {X 0,Y 455.869,Z 211.756,A -85,B 0,C 180,E1 -8491.094,E2 -8491.094} C_VEL
LIN {X 0,Y 455.329,Z 223.485,A -85,B 0,C 180,E1 -8492.023,E2 -8492.023} C_VEL
LIN {X 0,Y 454.826,Z 234.13,A -85,B 0,C 180,E1 -8493.086,E2 -8493.086} C_VEL
LIN {X 0,Y 454.302,Z 243.429,A -85,B 0,C 180,E1 -8494.243,E2 -8494.243} C_VEL
LIN {X 0,Y 453.786,Z 251.688,A -85,B 0,C 180,E1 -8495.505,E2 -8495.505} C_VEL
LIN {X 0,Y 453.385,Z 259.288,A -85,B 0,C 180,E1 -8496.959,E2 -8496.959} C_VEL
LIN {X 0,Y 453.094,Z 264.976,A -85,B 0,C 180,E1 -8498.348,E2 -8498.348} C_VEL
LIN {X 0,Y 452.799,Z 270.12,A -85,B 0,C 180,E1 -8499.999,E2 -8499.999} C_VEL
LIN {X 0,Y 452.655,Z 272.928,A -85,B 0,C 180,E1 -8501.249,E2 -8501.249} C_VEL
LIN {X 0,Y 452.59,Z 274.04,A -85,B 0,C 180,E1 -8501.891,E2 -8501.891} C_VEL
LIN {X 0,Y 452.534,Z 275.576,A -85,B 0,C 180,E1 -8503.119,E2 -8503.119} C_VEL
LIN {X 0,Y 452.468,Z 276.374,A -85,B 0,C 180,E1 -8504.397,E2 -8504.397} C_VEL
LIN {X 0,Y 452.473,Z 276.34,A -85,B 0,C 180,E1 -8505.656,E2 -8505.656} C_VEL
LIN {X 0,Y 452.502,Z 275.525,A -85,B 0,C 180,E1 -8506.891,E2 -8506.891} C_VEL
LIN {X 0,Y 452.594,Z 273.849,A -85,B 0,C 180,E1 -8508.189,E2 -8508.189} C_VEL
LIN {X 0,Y 452.751,Z 271.213,A -85,B 0,C 180,E1 -8509.518,E2 -8509.518} C_VEL
LIN {X 0,Y 452.917,Z 267.473,A -85,B 0,C 180,E1 -8510.882,E2 -8510.882} C_VEL
LIN {X 0,Y 453.19,Z 261.416,A -85,B 0,C 180,E1 -8512.532,E2 -8512.532} C_VEL
LIN {X 0,Y 453.52,Z 254.761,A -85,B 0,C 180,E1 -8513.923,E2 -8513.923} C_VEL
LIN {X 0,Y 453.916,Z 247.52,A -85,B 0,C 180,E1 -8515.144,E2 -8515.144} C_VEL
LIN {X 0,Y 454.463,Z 238.146,A -85,B 0,C 180,E1 -8516.427,E2 -8516.427} C_VEL
LIN {X 0,Y 454.927,Z 228.55,A -85,B 0,C 180,E1 -8517.494,E2 -8517.494} C_VEL
LIN {X 0,Y 455.433,Z 217.429,A -85,B 0,C 180,E1 -8518.483,E2 -8518.483} C_VEL
LIN {X 0,Y 455.925,Z 205.917,A -85,B 0,C 180,E1 -8519.295,E2 -8519.295} C_VEL
LIN {X 0,Y 456.439,Z 193.604,A -85,B 0,C 180,E1 -8519.957,E2 -8519.957} C_VEL
LIN {X 0,Y 456.268,Z 188.55,A -85,B 0,C 180,E1 -8520.186,E2 -8520.186} C_VEL
LIN {X 0,Y 453.164,Z 175.23,A -85,B 0,C 180,E1 -8520.738,E2 -8520.738} C_VEL
LIN {X 0,Y 452.684,Z 173.194,A -85,B 0,C 180,E1 -8520.818,E2 -8520.818} C_VEL
LIN {X 0,Y 452.795,Z 169.364,A -85,B 0,C 180,E1 -8524.24,E2 -8524.24} C_VEL
LIN {X 0,Y 452.753,Z 166.149,A -85,B 0,C 180,E1 -8527.165,E2 -8527.165} C_VEL
LIN {X 0,Y 452.786,Z 164.187,A -85,B 0,C 180,E1 -8528.965,E2 -8528.965} C_VEL
LIN {X 0,Y 452.156,Z 163.452,A -85,B 0,C 180,E1 -8529.702,E2 -8529.702} C_VEL
LIN {X 0,Y 449.337,Z 162.446,A -85,B 0,C 180,E1 -8530.904,E2 -8530.904} C_VEL
LIN {X 0,Y 446.934,Z 161.66,A -85,B 0,C 180,E1 -8531.874,E2 -8531.874} C_VEL
LIN {X 0,Y 445.904,Z 160.965,A -85,B 0,C 180,E1 -8532.621,E2 -8532.621} C_VEL
LIN {X 0,Y 445.821,Z 160.701,A -85,B 0,C 180,E1 -8532.874,E2 -8532.874} C_VEL
LIN {X 0,Y 445.908,Z 158.025,A -85,B 0,C 180,E1 -8535.393,E2 -8535.393} C_VEL
LIN {X 0,Y 445.941,Z 157.06,A -85,B 0,C 180,E1 -8536.326,E2 -8536.326} C_VEL
LIN {X 0,Y 446.297,Z 156.893,A -85,B 0,C 180,E1 -8539.107,E2 -8539.107} C_VEL
LIN {X 0,Y 446.565,Z 156.861,A -85,B 0,C 180,E1 -8541.857,E2 -8541.857} C_VEL
LIN {X 0,Y 446.637,Z 156.851,A -85,B 0,C 180,E1 -8544.582,E2 -8544.582} C_VEL
LIN {X 0,Y 446.706,Z 156.841,A -85,B 0,C 180,E1 -8547.295,E2 -8547.295} C_VEL
LIN {X 0,Y 446.791,Z 156.834,A -85,B 0,C 180,E1 -8550,E2 -8550} C_VEL
LIN {X 0,Y 446.706,Z 156.84,A -85,B 0,C 180,E1 -8552.705,E2 -8552.705} C_VEL
LIN {X 0,Y 446.635,Z 156.851,A -85,B 0,C 180,E1 -8556.324,E2 -8556.324} C_VEL
LIN {X 0,Y 446.535,Z 156.862,A -85,B 0,C 180,E1 -8559.055,E2 -8559.055} C_VEL
LIN {X 0,Y 446.518,Z 156.864,A -85,B 0,C 180,E1 -8562.73,E2 -8562.73} C_VEL
LIN {X 0,Y 446.493,Z 156.869,A -85,B 0,C 180,E1 -8566.228,E2 -8566.228} C_VEL
LIN {X 0,Y 446.466,Z 156.873,A -85,B 0,C 180,E1 -8569.303,E2 -8569.303} C_VEL
LIN {X 0,Y 446.415,Z 156.878,A -85,B 0,C 180,E1 -8572.2,E2 -8572.2} C_VEL
LIN {X 0,Y 446.455,Z 156.874,A -85,B 0,C 180,E1 -8575.152,E2 -8575.152} C_VEL
LIN {X 0,Y 446.481,Z 156.868,A -85,B 0,C 180,E1 -8578.179,E2 -8578.179} C_VEL
LIN {X 0,Y 446.416,Z 156.878,A -85,B 0,C 180,E1 -8581.775,E2 -8581.775} C_VEL
LIN {X 0,Y 446.425,Z 156.876,A -85,B 0,C 180,E1 -8584.523,E2 -8584.523} C_VEL
LIN {X 0,Y 446.413,Z 156.877,A -85,B 0,C 180,E1 -8588.08,E2 -8588.08} C_VEL
LIN {X 0,Y 446.424,Z 156.879,A -85,B 0,C 180,E1 -8590.918,E2 -8590.918} C_VEL
LIN {X 0,Y 446.42,Z 156.876,A -85,B 0,C 180,E1 -8593.844,E2 -8593.844} C_VEL
LIN {X 0,Y 446.397,Z 156.881,A -85,B 0,C 180,E1 -8596.404,E2 -8596.404} C_VEL
LIN {X 0,Y 446.425,Z 156.879,A -85,B 0,C 180,E1 -8599.083,E2 -8599.083} C_VEL
LIN {X 0,Y 446.426,Z 156.877,A -85,B 0,C 180,E1 -8602.124,E2 -8602.124} C_VEL
LIN {X 0,Y 446.427,Z 156.877,A -85,B 0,C 180,E1 -8605.477,E2 -8605.477} C_VEL
LIN {X 0,Y 446.414,Z 156.88,A -85,B 0,C 180,E1 -8608.7,E2 -8608.7} C_VEL
LIN {X 0,Y 446.484,Z 156.869,A -85,B 0,C 180,E1 -8611.822,E2 -8611.822} C_VEL
LIN {X 0,Y 446.457,Z 156.875,A -85,B 0,C 180,E1 -8614.848,E2 -8614.848} C_VEL
LIN {X 0,Y 446.448,Z 156.875,A -85,B 0,C 180,E1 -8618.246,E2 -8618.246} C_VEL
LIN {X 0,Y 446.452,Z 156.873,A -85,B 0,C 180,E1 -8621.649,E2 -8621.649} C_VEL
LIN {X 0,Y 446.508,Z 156.868,A -85,B 0,C 180,E1 -8624.48,E2 -8624.48} C_VEL
LIN {X 0,Y 446.519,Z 156.867,A -85,B 0,C 180,E1 -8628.194,E2 -8628.194} C_VEL
LIN {X 0,Y 446.535,Z 156.863,A -85,B 0,C 180,E1 -8630.945,E2 -8630.945} C_VEL
LIN {X 0,Y 446.642,Z 156.851,A -85,B 0,C 180,E1 -8633.677,E2 -8633.677} C_VEL
LIN {X 0,Y 446.71,Z 156.841,A -85,B 0,C 180,E1 -8637.295,E2 -8637.295} C_VEL
LIN {X 0,Y 446.795,Z 156.832,A -85,B 0,C 180,E1 -8640,E2 -8640} C_VEL
LIN {X 0,Y 446.693,Z 156.844,A -85,B 0,C 180,E1 -8642.706,E2 -8642.706} C_VEL
LIN {X 0,Y 446.623,Z 156.854,A -85,B 0,C 180,E1 -8646.324,E2 -8646.324} C_VEL
LIN {X 0,Y 446.523,Z 156.867,A -85,B 0,C 180,E1 -8649.97,E2 -8649.97} C_VEL
LIN {X 0,Y 446.524,Z 156.864,A -85,B 0,C 180,E1 -8652.73,E2 -8652.73} C_VEL
LIN {X 0,Y 446.498,Z 156.868,A -85,B 0,C 180,E1 -8656.228,E2 -8656.228} C_VEL
LIN {X 0,Y 446.472,Z 156.872,A -85,B 0,C 180,E1 -8659.304,E2 -8659.304} C_VEL
LIN {X 0,Y 446.42,Z 156.878,A -85,B 0,C 180,E1 -8662.2,E2 -8662.2} C_VEL
LIN {X 0,Y 446.46,Z 156.874,A -85,B 0,C 180,E1 -8665.153,E2 -8665.153} C_VEL
LIN {X 0,Y 446.487,Z 156.869,A -85,B 0,C 180,E1 -8668.179,E2 -8668.179} C_VEL
LIN {X 0,Y 446.421,Z 156.879,A -85,B 0,C 180,E1 -8671.775,E2 -8671.775} C_VEL
LIN {X 0,Y 446.425,Z 156.877,A -85,B 0,C 180,E1 -8674.524,E2 -8674.524} C_VEL
LIN {X 0,Y 446.417,Z 156.88,A -85,B 0,C 180,E1 -8678.079,E2 -8678.079} C_VEL
LIN {X 0,Y 446.429,Z 156.878,A -85,B 0,C 180,E1 -8680.918,E2 -8680.918} C_VEL
LIN {X 0,Y 446.404,Z 156.877,A -85,B 0,C 180,E1 -8683.846,E2 -8683.846} C_VEL
LIN {X 0,Y 446.4,Z 156.877,A -85,B 0,C 180,E1 -8686.404,E2 -8686.404} C_VEL
LIN {X 0,Y 446.466,Z 156.942,A -85,B 0,C 180,E1 -8688.085,E2 -8688.085} C_VEL
LIN {X 0,Y 447.641,Z 163.189,A -85,B 0,C 180,E1 -8691.097,E2 -8691.097} C_VEL
LIN {X 0,Y 448.399,Z 168.341,A -85,B 0,C 180,E1 -8693.445,E2 -8693.445} C_VEL
LIN {X 0,Y 448.294,Z 173.524,A -85,B 0,C 180,E1 -8695.641,E2 -8695.641} C_VEL
LIN {X 0,Y 447.825,Z 181.322,A -85,B 0,C 180,E1 -8698.809,E2 -8698.809} C_VEL
LIN {X 0,Y 447.292,Z 190.505,A -85,B 0,C 180,E1 -8702.386,E2 -8702.386} C_VEL
LIN {X 0,Y 446.814,Z 199.607,A -85,B 0,C 180,E1 -8705.825,E2 -8705.825} C_VEL
LIN {X 0,Y 446.456,Z 209.285,A -85,B 0,C 180,E1 -8709.256,E2 -8709.256} C_VEL
LIN {X 0,Y 446.176,Z 217.288,A -85,B 0,C 180,E1 -8712.112,E2 -8712.112} C_VEL
LIN {X 0,Y 446.037,Z 222.096,A -85,B 0,C 180,E1 -8713.819,E2 -8713.819} C_VEL
LIN {X 0,Y 448.487,Z 237.082,A -85,B 0,C 180,E1 -8714.344,E2 -8714.344} C_VEL
LIN {X 0,Y 449.422,Z 244.978,A -85,B 0,C 180,E1 -8714.699,E2 -8714.699} C_VEL
LIN {X 0,Y 448.948,Z 256.004,A -85,B 0,C 180,E1 -8715.263,E2 -8715.263} C_VEL
LIN {X 0,Y 448.371,Z 267.886,A -85,B 0,C 180,E1 -8716.055,E2 -8716.055} C_VEL
LIN {X 0,Y 447.799,Z 278.873,A -85,B 0,C 180,E1 -8716.993,E2 -8716.993} C_VEL
LIN {X 0,Y 447.309,Z 288.306,A -85,B 0,C 180,E1 -8717.984,E2 -8717.984} C_VEL
LIN {X 0,Y 446.699,Z 297.193,A -85,B 0,C 180,E1 -8719.117,E2 -8719.117} C_VEL
LIN {X 0,Y 446.26,Z 305.878,A -85,B 0,C 180,E1 -8720.482,E2 -8720.482} C_VEL
LIN {X 0,Y 445.885,Z 312.819,A -85,B 0,C 180,E1 -8721.845,E2 -8721.845} C_VEL
LIN {X 0,Y 445.65,Z 318.388,A -85,B 0,C 180,E1 -8723.208,E2 -8723.208} C_VEL
LIN {X 0,Y 445.54,Z 322.758,A -85,B 0,C 180,E1 -8724.569,E2 -8724.569} C_VEL
LIN {X 0,Y 445.428,Z 325.068,A -85,B 0,C 180,E1 -8725.475,E2 -8725.475} C_VEL
LIN {X 0,Y 445.397,Z 326.944,A -85,B 0,C 180,E1 -8726.381,E2 -8726.381} C_VEL
LIN {X 0,Y 445.423,Z 328.354,A -85,B 0,C 180,E1 -8727.287,E2 -8727.287} C_VEL
LIN {X 0,Y 445.356,Z 329.965,A -85,B 0,C 180,E1 -8729.096,E2 -8729.096} C_VEL
LIN {X 0,Y 445.35,Z 330.179,A -85,B 0,C 180,E1 -8730,E2 -8730} C_VEL
LIN {X 0,Y 445.356,Z 329.959,A -85,B 0,C 180,E1 -8730.904,E2 -8730.904} C_VEL
LIN {X 0,Y 445.423,Z 328.338,A -85,B 0,C 180,E1 -8732.713,E2 -8732.713} C_VEL
LIN {X 0,Y 445.398,Z 326.92,A -85,B 0,C 180,E1 -8733.619,E2 -8733.619} C_VEL
LIN {X 0,Y 445.501,Z 323.953,A -85,B 0,C 180,E1 -8734.978,E2 -8734.978} C_VEL
LIN {X 0,Y 445.588,Z 319.555,A -85,B 0,C 180,E1 -8736.451,E2 -8736.451} C_VEL
LIN {X 0,Y 445.805,Z 313.76,A -85,B 0,C 180,E1 -8737.929,E2 -8737.929} C_VEL
LIN {X 0,Y 446.182,Z 307.025,A -85,B 0,C 180,E1 -8739.291,E2 -8739.291} C_VEL
LIN {X 0,Y 446.619,Z 298.669,A -85,B 0,C 180,E1 -8740.655,E2 -8740.655} C_VEL
LIN {X 0,Y 447.172,Z 290.115,A -85,B 0,C 180,E1 -8741.79,E2 -8741.79} C_VEL
LIN {X 0,Y 447.71,Z 280.339,A -85,B 0,C 180,E1 -8742.85,E2 -8742.85} C_VEL
LIN {X 0,Y 448.256,Z 269.116,A -85,B 0,C 180,E1 -8743.833,E2 -8743.833} C_VEL
LIN {X 0,Y 448.826,Z 257.701,A -85,B 0,C 180,E1 -8744.625,E2 -8744.625} C_VEL
LIN {X 0,Y 449.375,Z 246.006,A -85,B 0,C 180,E1 -8745.245,E2 -8745.245} C_VEL
LIN {X 0,Y 448.737,Z 238.891,A -85,B 0,C 180,E1 -8745.567,E2 -8745.567} C_VEL
LIN {X 0,Y 446.65,Z 226.103,A -85,B 0,C 180,E1 -8746.045,E2 -8746.045} C_VEL
LIN {X 0,Y 446.008,Z 221.723,A -85,B 0,C 180,E1 -8746.182,E2 -8746.182} C_VEL
LIN {X 0,Y 446.329,Z 212.738,A -85,B 0,C 180,E1 -8749.31,E2 -8749.31} C_VEL
LIN {X 0,Y 446.59,Z 203.196,A -85,B 0,C 180,E1 -8752.679,E2 -8752.679} C_VEL
LIN {X 0,Y 446.923,Z 195.094,A -85,B 0,C 180,E1 -8755.623,E2 -8755.623} C_VEL
LIN {X 0,Y 447.352,Z 186.927,A -85,B 0,C 180,E1 -8758.712,E2 -8758.712} C_VEL
LIN {X 0,Y 447.821,Z 178.499,A -85,B 0,C 180,E1 -8762.063,E2 -8762.063} C_VEL
LIN {X 0,Y 448.415,Z 170.471,A -85,B 0,C 180,E1 -8765.444,E2 -8765.444} C_VEL
LIN {X 0,Y 448.305,Z 167.217,A -85,B 0,C 180,E1 -8766.915,E2 -8766.915} C_VEL
LIN {X 0,Y 447.143,Z 160.726,A -85,B 0,C 180,E1 -8770.123,E2 -8770.123} C_VEL
LIN {X 0,Y 446.438,Z 156.879,A -85,B 0,C 180,E1 -8772.277,E2 -8772.277} C_VEL
LIN {X 0,Y 446.458,Z 156.876,A -85,B 0,C 180,E1 -8775.103,E2 -8775.103} C_VEL
LIN {X 0,Y 446.432,Z 156.881,A -85,B 0,C 180,E1 -8778.609,E2 -8778.609} C_VEL
LIN {X 0,Y 446.464,Z 156.875,A -85,B 0,C 180,E1 -8780.975,E2 -8780.975} C_VEL
LIN {X 0,Y 446.424,Z 156.879,A -85,B 0,C 180,E1 -8784.374,E2 -8784.374} C_VEL
LIN {X 0,Y 446.427,Z 156.878,A -85,B 0,C 180,E1 -8787.638,E2 -8787.638} C_VEL
LIN {X 0,Y 446.454,Z 156.874,A -85,B 0,C 180,E1 -8790.791,E2 -8790.791} C_VEL
LIN {X 0,Y 446.482,Z 156.871,A -85,B 0,C 180,E1 -8793.848,E2 -8793.848} C_VEL
LIN {X 0,Y 446.433,Z 156.877,A -85,B 0,C 180,E1 -8796.823,E2 -8796.823} C_VEL
LIN {X 0,Y 446.448,Z 156.874,A -85,B 0,C 180,E1 -8799.737,E2 -8799.737} C_VEL
LIN {X 0,Y 446.461,Z 156.874,A -85,B 0,C 180,E1 -8802.597,E2 -8802.597} C_VEL
LIN {X 0,Y 446.475,Z 156.873,A -85,B 0,C 180,E1 -8805.412,E2 -8805.412} C_VEL
LIN {X 0,Y 446.522,Z 156.866,A -85,B 0,C 180,E1 -8808.193,E2 -8808.193} C_VEL
LIN {X 0,Y 446.605,Z 156.856,A -85,B 0,C 180,E1 -8811.857,E2 -8811.857} C_VEL
LIN {X 0,Y 446.65,Z 156.852,A -85,B 0,C 180,E1 -8814.582,E2 -8814.582} C_VEL
LIN {X 0,Y 446.713,Z 156.842,A -85,B 0,C 180,E1 -8817.294,E2 -8817.294} C_VEL
LIN {X 0,Y 446.799,Z 156.832,A -85,B 0,C 180,E1 -8820,E2 -8820} C_VEL
LIN {X 0,Y 446.712,Z 156.843,A -85,B 0,C 180,E1 -8822.705,E2 -8822.705} C_VEL
LIN {X 0,Y 446.65,Z 156.853,A -85,B 0,C 180,E1 -8826.323,E2 -8826.323} C_VEL
LIN {X 0,Y 446.496,Z 156.871,A -85,B 0,C 180,E1 -8829.056,E2 -8829.056} C_VEL
LIN {X 0,Y 446.265,Z 156.903,A -85,B 0,C 180,E1 -8830.893,E2 -8830.893} C_VEL
LIN {X 0,Y 446.253,Z 157.979,A -85,B 0,C 180,E1 -8832.462,E2 -8832.462} C_VEL
LIN {X 0,Y 446.113,Z 161.56,A -85,B 0,C 180,E1 -8836.056,E2 -8836.056} C_VEL
LIN {X 0,Y 445.948,Z 164.863,A -85,B 0,C 180,E1 -8839.326,E2 -8839.326} C_VEL
LIN {X 0,Y 445.868,Z 167.851,A -85,B 0,C 180,E1 -8842.228,E2 -8842.228} C_VEL
LIN {X 0,Y 445.807,Z 170.908,A -85,B 0,C 180,E1 -8845.191,E2 -8845.191} C_VEL
LIN {X 0,Y 445.799,Z 174.605,A -85,B 0,C 180,E1 -8848.739,E2 -8848.739} C_VEL
LIN {X 0,Y 445.784,Z 174.849,A -85,B 0,C 180,E1 -8848.966,E2 -8848.966} C_VEL
LIN {X 0,Y 449.474,Z 189.716,A -85,B 0,C 180,E1 -8849.619,E2 -8849.619} C_VEL
LIN {X 0,Y 449.771,Z 193.633,A -85,B 0,C 180,E1 -8849.807,E2 -8849.807} C_VEL
LIN {X 0,Y 449.345,Z 205.065,A -85,B 0,C 180,E1 -8850.408,E2 -8850.408} C_VEL
LIN {X 0,Y 448.848,Z 215.471,A -85,B 0,C 180,E1 -8851.111,E2 -8851.111} C_VEL
LIN {X 0,Y 448.333,Z 226.554,A -85,B 0,C 180,E1 -8852.062,E2 -8852.062} C_VEL
LIN {X 0,Y 447.75,Z 237.071,A -85,B 0,C 180,E1 -8853.189,E2 -8853.189} C_VEL
LIN {X 0,Y 447.203,Z 246.552,A -85,B 0,C 180,E1 -8854.454,E2 -8854.454} C_VEL
LIN {X 0,Y 446.603,Z 254.902,A -85,B 0,C 180,E1 -8855.849,E2 -8855.849} C_VEL
LIN {X 0,Y 446.273,Z 261.896,A -85,B 0,C 180,E1 -8857.322,E2 -8857.322} C_VEL
LIN {X 0,Y 445.984,Z 266.41,A -85,B 0,C 180,E1 -8858.52,E2 -8858.52} C_VEL
LIN {X 0,Y 445.768,Z 270.295,A -85,B 0,C 180,E1 -8859.816,E2 -8859.816} C_VEL
LIN {X 0,Y 445.563,Z 273.933,A -85,B 0,C 180,E1 -8861.488,E2 -8861.488} C_VEL
LIN {X 0,Y 445.459,Z 275.65,A -85,B 0,C 180,E1 -8862.719,E2 -8862.719} C_VEL
LIN {X 0,Y 445.393,Z 276.627,A -85,B 0,C 180,E1 -8863.97,E2 -8863.97} C_VEL
LIN {X 0,Y 445.366,Z 276.858,A -85,B 0,C 180,E1 -8865.243,E2 -8865.243} C_VEL
LIN {X 0,Y 445.397,Z 276.296,A -85,B 0,C 180,E1 -8866.538,E2 -8866.538} C_VEL
LIN {X 0,Y 445.475,Z 274.858,A -85,B 0,C 180,E1 -8867.858,E2 -8867.858} C_VEL
LIN {X 0,Y 445.625,Z 272.487,A -85,B 0,C 180,E1 -8869.201,E2 -8869.201} C_VEL
LIN {X 0,Y 445.843,Z 268.071,A -85,B 0,C 180,E1 -8870.91,E2 -8870.91} C_VEL
LIN {X 0,Y 446.105,Z 262.894,A -85,B 0,C 180,E1 -8872.376,E2 -8872.376} C_VEL
LIN {X 0,Y 446.46,Z 255.966,A -85,B 0,C 180,E1 -8873.903,E2 -8873.903} C_VEL
LIN {X 0,Y 446.895,Z 248.478,A -85,B 0,C 180,E1 -8875.209,E2 -8875.209} C_VEL
LIN {X 0,Y 447.434,Z 239.75,A -85,B 0,C 180,E1 -8876.443,E2 -8876.443} C_VEL
LIN {X 0,Y 447.964,Z 229.42,A -85,B 0,C 180,E1 -8877.63,E2 -8877.63} C_VEL
LIN {X 0,Y 448.491,Z 218.882,A -85,B 0,C 180,E1 -8878.598,E2 -8878.598} C_VEL
LIN {X 0,Y 448.966,Z 207.609,A -85,B 0,C 180,E1 -8879.423,E2 -8879.423} C_VEL
LIN {X 0,Y 449.534,Z 195.693,A -85,B 0,C 180,E1 -8880.095,E2 -8880.095} C_VEL
LIN {X 0,Y 449.61,Z 190.943,A -85,B 0,C 180,E1 -8880.315,E2 -8880.315} C_VEL
LIN {X 0,Y 446.807,Z 178.411,A -85,B 0,C 180,E1 -8880.881,E2 -8880.881} C_VEL
LIN {X 0,Y 445.629,Z 173.584,A -85,B 0,C 180,E1 -8881.055,E2 -8881.055} C_VEL
LIN {X 0,Y 445.711,Z 170.305,A -85,B 0,C 180,E1 -8883.997,E2 -8883.997} C_VEL
LIN {X 0,Y 445.704,Z 167.257,A -85,B 0,C 180,E1 -8886.783,E2 -8886.783} C_VEL
LIN {X 0,Y 445.729,Z 164.097,A -85,B 0,C 180,E1 -8889.703,E2 -8889.703} C_VEL
LIN {X 0,Y 445.829,Z 161.026,A -85,B 0,C 180,E1 -8892.571,E2 -8892.571} C_VEL
LIN {X 0,Y 445.821,Z 160.701,A -85,B 0,C 180,E1 -8892.874,E2 -8892.874} C_VEL
LIN {X 0,Y 445.154,Z 159.971,A -85,B 0,C 180,E1 -8893.622,E2 -8893.622} C_VEL
LIN {X 0,Y 442.309,Z 158.998,A -85,B 0,C 180,E1 -8894.841,E2 -8894.841} C_VEL
LIN {X 0,Y 439.948,Z 158.322,A -85,B 0,C 180,E1 -8895.828,E2 -8895.828} C_VEL
LIN {X 0,Y 438.998,Z 157.944,A -85,B 0,C 180,E1 -8896.591,E2 -8896.591} C_VEL
LIN {X 0,Y 438.955,Z 157.86,A -85,B 0,C 180,E1 -8896.849,E2 -8896.849} C_VEL
LIN {X 0,Y 439.235,Z 157.773,A -85,B 0,C 180,E1 -8898.93,E2 -8898.93} C_VEL
LIN {X 0,Y 439.521,Z 157.738,A -85,B 0,C 180,E1 -8901.726,E2 -8901.726} C_VEL
LIN {X 0,Y 439.611,Z 157.727,A -85,B 0,C 180,E1 -8904.495,E2 -8904.495} C_VEL
LIN {X 0,Y 439.634,Z 157.724,A -85,B 0,C 180,E1 -8908.168,E2 -8908.168} C_VEL
LIN {X 0,Y 439.761,Z 157.71,A -85,B 0,C 180,E1 -8910,E2 -8910} C_VEL
LIN {X 0,Y 439.653,Z 157.719,A -85,B 0,C 180,E1 -8912.749,E2 -8912.749} C_VEL
LIN {X 0,Y 439.61,Z 157.726,A -85,B 0,C 180,E1 -8916.425,E2 -8916.425} C_VEL
LIN {X 0,Y 439.496,Z 157.739,A -85,B 0,C 180,E1 -8919.202,E2 -8919.202} C_VEL
LIN {X 0,Y 439.462,Z 157.743,A -85,B 0,C 180,E1 -8922.938,E2 -8922.938} C_VEL
LIN {X 0,Y 439.444,Z 157.747,A -85,B 0,C 180,E1 -8926.349,E2 -8926.349} C_VEL
LIN {X 0,Y 439.399,Z 157.754,A -85,B 0,C 180,E1 -8929.626,E2 -8929.626} C_VEL
LIN {X 0,Y 439.362,Z 157.756,A -85,B 0,C 180,E1 -8932.576,E2 -8932.576} C_VEL
LIN {X 0,Y 439.402,Z 157.753,A -85,B 0,C 180,E1 -8935.585,E2 -8935.585} C_VEL
LIN {X 0,Y 439.414,Z 157.749,A -85,B 0,C 180,E1 -8938.674,E2 -8938.674} C_VEL
LIN {X 0,Y 439.367,Z 157.756,A -85,B 0,C 180,E1 -8942.031,E2 -8942.031} C_VEL
LIN {X 0,Y 439.391,Z 157.755,A -85,B 0,C 180,E1 -8945.341,E2 -8945.341} C_VEL
LIN {X 0,Y 439.38,Z 157.755,A -85,B 0,C 180,E1 -8948.595,E2 -8948.595} C_VEL
LIN {X 0,Y 439.386,Z 157.755,A -85,B 0,C 180,E1 -8951.257,E2 -8951.257} C_VEL
LIN {X 0,Y 439.403,Z 157.753,A -85,B 0,C 180,E1 -8954.729,E2 -8954.729} C_VEL
LIN {X 0,Y 439.394,Z 157.752,A -85,B 0,C 180,E1 -8957.796,E2 -8957.796} C_VEL
LIN {X 0,Y 439.428,Z 157.747,A -85,B 0,C 180,E1 -8960.228,E2 -8960.228} C_VEL
LIN {X 0,Y 439.375,Z 157.754,A -85,B 0,C 180,E1 -8963.714,E2 -8963.714} C_VEL
LIN {X 0,Y 439.37,Z 157.757,A -85,B 0,C 180,E1 -8967.054,E2 -8967.054} C_VEL
LIN {X 0,Y 439.381,Z 157.755,A -85,B 0,C 180,E1 -8970.275,E2 -8970.275} C_VEL
LIN {X 0,Y 439.428,Z 157.748,A -85,B 0,C 180,E1 -8973.397,E2 -8973.397} C_VEL
LIN {X 0,Y 439.386,Z 157.756,A -85,B 0,C 180,E1 -8976.43,E2 -8976.43} C_VEL
LIN {X 0,Y 439.388,Z 157.752,A -85,B 0,C 180,E1 -8979.398,E2 -8979.398} C_VEL
LIN {X 0,Y 439.426,Z 157.751,A -85,B 0,C 180,E1 -8982.31,E2 -8982.31} C_VEL
LIN {X 0,Y 439.448,Z 157.744,A -85,B 0,C 180,E1 -8985.174,E2 -8985.174} C_VEL
LIN {X 0,Y 439.485,Z 157.742,A -85,B 0,C 180,E1 -8988.002,E2 -8988.002} C_VEL
LIN {X 0,Y 439.532,Z 157.735,A -85,B 0,C 180,E1 -8991.726,E2 -8991.726} C_VEL
LIN {X 0,Y 439.621,Z 157.726,A -85,B 0,C 180,E1 -8994.496,E2 -8994.496} C_VEL
LIN {X 0,Y 439.636,Z 157.725,A -85,B 0,C 180,E1 -8998.168,E2 -8998.168} C_VEL
LIN {X 0,Y 439.764,Z 157.708,A -85,B 0,C 180,E1 -9000,E2 -9000} C_VEL
LIN {X 0,Y 439.642,Z 157.722,A -85,B 0,C 180,E1 -9002.749,E2 -9002.749} C_VEL
LIN {X 0,Y 439.595,Z 157.729,A -85,B 0,C 180,E1 -9006.426,E2 -9006.426} C_VEL
LIN {X 0,Y 439.497,Z 157.74,A -85,B 0,C 180,E1 -9009.202,E2 -9009.202} C_VEL
LIN {X 0,Y 439.468,Z 157.743,A -85,B 0,C 180,E1 -9012.938,E2 -9012.938} C_VEL
LIN {X 0,Y 439.449,Z 157.745,A -85,B 0,C 180,E1 -9016.349,E2 -9016.349} C_VEL
LIN {X 0,Y 439.405,Z 157.754,A -85,B 0,C 180,E1 -9019.627,E2 -9019.627} C_VEL
LIN {X 0,Y 439.367,Z 157.755,A -85,B 0,C 180,E1 -9022.576,E2 -9022.576} C_VEL
LIN {X 0,Y 439.408,Z 157.753,A -85,B 0,C 180,E1 -9025.585,E2 -9025.585} C_VEL
LIN {X 0,Y 439.42,Z 157.749,A -85,B 0,C 180,E1 -9028.674,E2 -9028.674} C_VEL
LIN {X 0,Y 439.371,Z 157.755,A -85,B 0,C 180,E1 -9032.03,E2 -9032.03} C_VEL
LIN {X 0,Y 439.394,Z 157.755,A -85,B 0,C 180,E1 -9035.34,E2 -9035.34} C_VEL
LIN {X 0,Y 439.379,Z 157.754,A -85,B 0,C 180,E1 -9038.596,E2 -9038.596} C_VEL
LIN {X 0,Y 439.391,Z 157.755,A -85,B 0,C 180,E1 -9041.257,E2 -9041.257} C_VEL
LIN {X 0,Y 439.404,Z 157.748,A -85,B 0,C 180,E1 -9044.729,E2 -9044.729} C_VEL
LIN {X 0,Y 439.426,Z 157.908,A -85,B 0,C 180,E1 -9047.799,E2 -9047.799} C_VEL
LIN {X 0,Y 440.624,Z 164.245,A -85,B 0,C 180,E1 -9050.911,E2 -9050.911} C_VEL
LIN {X 0,Y 441.431,Z 169.51,A -85,B 0,C 180,E1 -9053.358,E2 -9053.358} C_VEL
LIN {X 0,Y 441.323,Z 174.512,A -85,B 0,C 180,E1 -9055.52,E2 -9055.52} C_VEL
LIN {X 0,Y 440.809,Z 182.442,A -85,B 0,C 180,E1 -9058.791,E2 -9058.791} C_VEL
LIN {X 0,Y 440.254,Z 191.602,A -85,B 0,C 180,E1 -9062.423,E2 -9062.423} C_VEL
LIN {X 0,Y 439.813,Z 199.964,A -85,B 0,C 180,E1 -9065.621,E2 -9065.621} C_VEL
LIN {X 0,Y 439.434,Z 208.889,A -85,B 0,C 180,E1 -9068.909,E2 -9068.909} C_VEL
LIN {X 0,Y 439.126,Z 216.891,A -85,B 0,C 180,E1 -9071.815,E2 -9071.815} C_VEL
LIN {X 0,Y 438.989,Z 221.962,A -85,B 0,C 180,E1 -9073.575,E2 -9073.575} C_VEL
LIN {X 0,Y 441.222,Z 235.554,A -85,B 0,C 180,E1 -9074.037,E2 -9074.037} C_VEL
LIN {X 0,Y 442.515,Z 245.855,A -85,B 0,C 180,E1 -9074.513,E2 -9074.513} C_VEL
LIN {X 0,Y 441.959,Z 257.515,A -85,B 0,C 180,E1 -9075.142,E2 -9075.142} C_VEL
LIN {X 0,Y 441.363,Z 268.902,A -85,B 0,C 180,E1 -9075.946,E2 -9075.946} C_VEL
LIN {X 0,Y 440.734,Z 280.285,A -85,B 0,C 180,E1 -9076.963,E2 -9076.963} C_VEL
LIN {X 0,Y 440.208,Z 289.842,A -85,B 0,C 180,E1 -9078.021,E2 -9078.021} C_VEL
LIN {X 0,Y 439.609,Z 298.373,A -85,B 0,C 180,E1 -9079.173,E2 -9079.173} C_VEL
LIN {X 0,Y 439.153,Z 306.704,A -85,B 0,C 180,E1 -9080.559,E2 -9080.559} C_VEL
LIN {X 0,Y 438.752,Z 313.419,A -85,B 0,C 180,E1 -9081.943,E2 -9081.943} C_VEL
LIN {X 0,Y 438.527,Z 319.577,A -85,B 0,C 180,E1 -9083.559,E2 -9083.559} C_VEL
LIN {X 0,Y 438.435,Z 323.579,A -85,B 0,C 180,E1 -9084.942,E2 -9084.942} C_VEL
LIN {X 0,Y 438.302,Z 326.529,A -85,B 0,C 180,E1 -9086.323,E2 -9086.323} C_VEL
LIN {X 0,Y 438.351,Z 327.94,A -85,B 0,C 180,E1 -9087.243,E2 -9087.243} C_VEL
LIN {X 0,Y 438.269,Z 329.548,A -85,B 0,C 180,E1 -9089.081,E2 -9089.081} C_VEL
LIN {X 0,Y 438.29,Z 329.763,A -85,B 0,C 180,E1 -9090,E2 -9090} C_VEL
LIN {X 0,Y 438.269,Z 329.539,A -85,B 0,C 180,E1 -9090.919,E2 -9090.919} C_VEL
LIN {X 0,Y 438.351,Z 327.913,A -85,B 0,C 180,E1 -9092.757,E2 -9092.757} C_VEL
LIN {X 0,Y 438.303,Z 326.491,A -85,B 0,C 180,E1 -9093.678,E2 -9093.678} C_VEL
LIN {X 0,Y 438.435,Z 323.52,A -85,B 0,C 180,E1 -9095.058,E2 -9095.058} C_VEL
LIN {X 0,Y 438.507,Z 319.494,A -85,B 0,C 180,E1 -9096.442,E2 -9096.442} C_VEL
LIN {X 0,Y 438.754,Z 313.314,A -85,B 0,C 180,E1 -9098.057,E2 -9098.057} C_VEL
LIN {X 0,Y 439.142,Z 306.571,A -85,B 0,C 180,E1 -9099.442,E2 -9099.442} C_VEL
LIN {X 0,Y 439.6,Z 298.207,A -85,B 0,C 180,E1 -9100.828,E2 -9100.828} C_VEL
LIN {X 0,Y 440.183,Z 289.647,A -85,B 0,C 180,E1 -9101.98,E2 -9101.98} C_VEL
LIN {X 0,Y 440.737,Z 280.098,A -85,B 0,C 180,E1 -9103.033,E2 -9103.033} C_VEL
LIN {X 0,Y 441.319,Z 268.639,A -85,B 0,C 180,E1 -9104.055,E2 -9104.055} C_VEL
LIN {X 0,Y 441.96,Z 257.226,A -85,B 0,C 180,E1 -9104.858,E2 -9104.858} C_VEL
LIN {X 0,Y 442.503,Z 245.528,A -85,B 0,C 180,E1 -9105.487,E2 -9105.487} C_VEL
LIN {X 0,Y 440.863,Z 233.678,A -85,B 0,C 180,E1 -9106.026,E2 -9106.026} C_VEL
LIN {X 0,Y 438.91,Z 221.245,A -85,B 0,C 180,E1 -9106.454,E2 -9106.454} C_VEL
LIN {X 0,Y 439.259,Z 212.269,A -85,B 0,C 180,E1 -9109.633,E2 -9109.633} C_VEL
LIN {X 0,Y 439.561,Z 202.837,A -85,B 0,C 180,E1 -9113.062,E2 -9113.062} C_VEL
LIN {X 0,Y 439.934,Z 194.831,A -85,B 0,C 180,E1 -9116.061,E2 -9116.061} C_VEL
LIN {X 0,Y 440.36,Z 186.898,A -85,B 0,C 180,E1 -9119.129,E2 -9119.129} C_VEL
LIN {X 0,Y 440.866,Z 179.015,A -85,B 0,C 180,E1 -9122.339,E2 -9122.339} C_VEL
LIN {X 0,Y 441.342,Z 172.848,A -85,B 0,C 180,E1 -9124.979,E2 -9124.979} C_VEL
LIN {X 0,Y 441.39,Z 169.163,A -85,B 0,C 180,E1 -9126.646,E2 -9126.646} C_VEL
LIN {X 0,Y 440.359,Z 163.085,A -85,B 0,C 180,E1 -9129.672,E2 -9129.672} C_VEL
LIN {X 0,Y 439.386,Z 157.753,A -85,B 0,C 180,E1 -9132.627,E2 -9132.627} C_VEL
LIN {X 0,Y 439.406,Z 157.756,A -85,B 0,C 180,E1 -9135.271,E2 -9135.271} C_VEL
LIN {X 0,Y 439.393,Z 157.758,A -85,B 0,C 180,E1 -9138.743,E2 -9138.743} C_VEL
LIN {X 0,Y 439.382,Z 157.758,A -85,B 0,C 180,E1 -9141.607,E2 -9141.607} C_VEL
LIN {X 0,Y 439.403,Z 157.754,A -85,B 0,C 180,E1 -9144.844,E2 -9144.844} C_VEL
LIN {X 0,Y 439.378,Z 157.756,A -85,B 0,C 180,E1 -9148.139,E2 -9148.139} C_VEL
LIN {X 0,Y 439.437,Z 157.749,A -85,B 0,C 180,E1 -9151.598,E2 -9151.598} C_VEL
LIN {X 0,Y 439.41,Z 157.753,A -85,B 0,C 180,E1 -9154.415,E2 -9154.415} C_VEL
LIN {X 0,Y 439.37,Z 157.756,A -85,B 0,C 180,E1 -9157.424,E2 -9157.424} C_VEL
LIN {X 0,Y 439.445,Z 157.749,A -85,B 0,C 180,E1 -9160.663,E2 -9160.663} C_VEL
LIN {X 0,Y 439.467,Z 157.745,A -85,B 0,C 180,E1 -9164.224,E2 -9164.224} C_VEL
LIN {X 0,Y 439.488,Z 157.742,A -85,B 0,C 180,E1 -9168.001,E2 -9168.001} C_VEL
LIN {X 0,Y 439.553,Z 157.735,A -85,B 0,C 180,E1 -9171.726,E2 -9171.726} C_VEL
LIN {X 0,Y 439.626,Z 157.726,A -85,B 0,C 180,E1 -9174.495,E2 -9174.495} C_VEL
LIN {X 0,Y 439.641,Z 157.723,A -85,B 0,C 180,E1 -9178.167,E2 -9178.167} C_VEL
LIN {X 0,Y 439.769,Z 157.708,A -85,B 0,C 180,E1 -9180,E2 -9180} C_VEL
LIN {X 0,Y 439.659,Z 157.722,A -85,B 0,C 180,E1 -9182.748,E2 -9182.748} C_VEL
LIN {X 0,Y 439.621,Z 157.729,A -85,B 0,C 180,E1 -9186.425,E2 -9186.425} C_VEL
LIN {X 0,Y 439.447,Z 157.748,A -85,B 0,C 180,E1 -9189.202,E2 -9189.202} C_VEL
LIN {X 0,Y 439.205,Z 157.783,A -85,B 0,C 180,E1 -9191.07,E2 -9191.07} C_VEL
LIN {X 0,Y 439.178,Z 159.395,A -85,B 0,C 180,E1 -9192.946,E2 -9192.946} C_VEL
LIN {X 0,Y 439.075,Z 162.542,A -85,B 0,C 180,E1 -9196.18,E2 -9196.18} C_VEL
LIN {X 0,Y 438.874,Z 166.064,A -85,B 0,C 180,E1 -9199.65,E2 -9199.65} C_VEL
LIN {X 0,Y 438.802,Z 169.06,A -85,B 0,C 180,E1 -9202.605,E2 -9202.605} C_VEL
LIN {X 0,Y 438.73,Z 172.137,A -85,B 0,C 180,E1 -9205.627,E2 -9205.627} C_VEL
LIN {X 0,Y 438.743,Z 175.322,A -85,B 0,C 180,E1 -9208.701,E2 -9208.701} C_VEL
LIN {X 0,Y 442.239,Z 189.343,A -85,B 0,C 180,E1 -9209.318,E2 -9209.318} C_VEL
LIN {X 0,Y 442.995,Z 193.296,A -85,B 0,C 180,E1 -9209.524,E2 -9209.524} C_VEL
LIN {X 0,Y 442.474,Z 206.321,A -85,B 0,C 180,E1 -9210.218,E2 -9210.218} C_VEL
LIN {X 0,Y 441.859,Z 218.436,A -85,B 0,C 180,E1 -9211.087,E2 -9211.087} C_VEL
LIN {X 0,Y 441.313,Z 229.026,A -85,B 0,C 180,E1 -9212.051,E2 -9212.051} C_VEL
LIN {X 0,Y 440.777,Z 238.38,A -85,B 0,C 180,E1 -9213.099,E2 -9213.099} C_VEL
LIN {X 0,Y 440.271,Z 246.739,A -85,B 0,C 180,E1 -9214.242,E2 -9214.242} C_VEL
LIN {X 0,Y 439.654,Z 254.636,A -85,B 0,C 180,E1 -9215.563,E2 -9215.563} C_VEL
LIN {X 0,Y 439.257,Z 262.049,A -85,B 0,C 180,E1 -9217.126,E2 -9217.126} C_VEL
LIN {X 0,Y 438.913,Z 267.624,A -85,B 0,C 180,E1 -9218.643,E2 -9218.643} C_VEL
LIN {X 0,Y 438.689,Z 271.069,A -85,B 0,C 180,E1 -9219.852,E2 -9219.852} C_VEL
LIN {X 0,Y 438.535,Z 273.827,A -85,B 0,C 180,E1 -9221.129,E2 -9221.129} C_VEL
LIN {X 0,Y 438.383,Z 275.862,A -85,B 0,C 180,E1 -9222.484,E2 -9222.484} C_VEL
LIN {X 0,Y 438.313,Z 276.999,A -85,B 0,C 180,E1 -9223.818,E2 -9223.818} C_VEL
LIN {X 0,Y 438.278,Z 277.313,A -85,B 0,C 180,E1 -9225.125,E2 -9225.125} C_VEL
LIN {X 0,Y 438.314,Z 276.82,A -85,B 0,C 180,E1 -9226.412,E2 -9226.412} C_VEL
LIN {X 0,Y 438.391,Z 275.557,A -85,B 0,C 180,E1 -9227.676,E2 -9227.676} C_VEL
LIN {X 0,Y 438.612,Z 272.305,A -85,B 0,C 180,E1 -9229.538,E2 -9229.538} C_VEL
LIN {X 0,Y 438.772,Z 269.058,A -85,B 0,C 180,E1 -9230.809,E2 -9230.809} C_VEL
LIN {X 0,Y 438.981,Z 264.751,A -85,B 0,C 180,E1 -9232.112,E2 -9232.112} C_VEL
LIN {X 0,Y 439.292,Z 259.329,A -85,B 0,C 180,E1 -9233.422,E2 -9233.422} C_VEL
LIN {X 0,Y 439.702,Z 251.818,A -85,B 0,C 180,E1 -9234.872,E2 -9234.872} C_VEL
LIN {X 0,Y 440.251,Z 243.874,A -85,B 0,C 180,E1 -9236.109,E2 -9236.109} C_VEL
LIN {X 0,Y 440.761,Z 234.503,A -85,B 0,C 180,E1 -9237.306,E2 -9237.306} C_VEL
LIN {X 0,Y 441.348,Z 223.643,A -85,B 0,C 180,E1 -9238.419,E2 -9238.419} C_VEL
LIN {X 0,Y 441.917,Z 211.411,A -85,B 0,C 180,E1 -9239.408,E2 -9239.408} C_VEL
LIN {X 0,Y 442.492,Z 200.177,A -85,B 0,C 180,E1 -9240.111,E2 -9240.111} C_VEL
LIN {X 0,Y 442.707,Z 191.921,A -85,B 0,C 180,E1 -9240.519,E2 -9240.519} C_VEL
LIN {X 0,Y 439.91,Z 179.519,A -85,B 0,C 180,E1 -9241.1,E2 -9241.1} C_VEL
LIN {X 0,Y 438.57,Z 173.944,A -85,B 0,C 180,E1 -9241.324,E2 -9241.324} C_VEL
LIN {X 0,Y 438.651,Z 170.58,A -85,B 0,C 180,E1 -9244.368,E2 -9244.368} C_VEL
LIN {X 0,Y 438.63,Z 167.307,A -85,B 0,C 180,E1 -9247.384,E2 -9247.384} C_VEL
LIN {X 0,Y 438.755,Z 163.505,A -85,B 0,C 180,E1 -9250.919,E2 -9250.919} C_VEL
LIN {X 0,Y 438.856,Z 160.039,A -85,B 0,C 180,E1 -9254.202,E2 -9254.202} C_VEL
LIN {X 0,Y 438.874,Z 158.067,A -85,B 0,C 180,E1 -9256.101,E2 -9256.101} C_VEL
LIN {X 0,Y 438.955,Z 157.86,A -85,B 0,C 180,E1 -9256.849,E2 -9256.849} C_VEL
LIN {X 0,Y 438.41,Z 157.877,A -85,B 0,C 180,E1 -9257.615,E2 -9257.615} C_VEL
LIN {X 0,Y 435.728,Z 158.21,A -85,B 0,C 180,E1 -9258.865,E2 -9258.865} C_VEL
LIN {X 0,Y 433.423,Z 158.509,A -85,B 0,C 180,E1 -9259.873,E2 -9259.873} C_VEL
LIN {X 0,Y 432.457,Z 158.618,A -85,B 0,C 180,E1 -9260.651,E2 -9260.651} C_VEL
LIN {X 0,Y 432.394,Z 158.623,A -85,B 0,C 180,E1 -9260.914,E2 -9260.914} C_VEL
LIN {X 0,Y 432.548,Z 158.604,A -85,B 0,C 180,E1 -9263.469,E2 -9263.469} C_VEL
LIN {X 0,Y 432.396,Z 158.624,A -85,B 0,C 180,E1 -9265.338,E2 -9265.338} C_VEL
LIN {X 0,Y 432.604,Z 158.6,A -85,B 0,C 180,E1 -9268.138,E2 -9268.138} C_VEL
LIN {X 0,Y 432.731,Z 158.586,A -85,B 0,C 180,E1 -9270,E2 -9270} C_VEL
LIN {X 0,Y 432.602,Z 158.597,A -85,B 0,C 180,E1 -9272.793,E2 -9272.793} C_VEL
LIN {X 0,Y 432.565,Z 158.603,A -85,B 0,C 180,E1 -9276.53,E2 -9276.53} C_VEL
LIN {X 0,Y 432.439,Z 158.619,A -85,B 0,C 180,E1 -9279.353,E2 -9279.353} C_VEL
LIN {X 0,Y 432.427,Z 158.619,A -85,B 0,C 180,E1 -9282.803,E2 -9282.803} C_VEL
LIN {X 0,Y 432.409,Z 158.622,A -85,B 0,C 180,E1 -9286.479,E2 -9286.479} C_VEL
LIN {X 0,Y 432.336,Z 158.633,A -85,B 0,C 180,E1 -9289.96,E2 -9289.96} C_VEL
LIN {X 0,Y 432.316,Z 158.635,A -85,B 0,C 180,E1 -9292.964,E2 -9292.964} C_VEL
LIN {X 0,Y 432.361,Z 158.629,A -85,B 0,C 180,E1 -9296.033,E2 -9296.033} C_VEL
LIN {X 0,Y 432.34,Z 158.634,A -85,B 0,C 180,E1 -9299.188,E2 -9299.188} C_VEL
LIN {X 0,Y 432.32,Z 158.633,A -85,B 0,C 180,E1 -9302.443,E2 -9302.443} C_VEL
LIN {X 0,Y 432.341,Z 158.632,A -85,B 0,C 180,E1 -9305.632,E2 -9305.632} C_VEL
LIN {X 0,Y 432.347,Z 158.632,A -85,B 0,C 180,E1 -9309.343,E2 -9309.343} C_VEL
LIN {X 0,Y 432.331,Z 158.632,A -85,B 0,C 180,E1 -9311.797,E2 -9311.797} C_VEL
LIN {X 0,Y 432.337,Z 158.63,A -85,B 0,C 180,E1 -9314.347,E2 -9314.347} C_VEL
LIN {X 0,Y 432.318,Z 158.637,A -85,B 0,C 180,E1 -9317.016,E2 -9317.016} C_VEL
LIN {X 0,Y 432.334,Z 158.631,A -85,B 0,C 180,E1 -9319.821,E2 -9319.821} C_VEL
LIN {X 0,Y 432.314,Z 158.637,A -85,B 0,C 180,E1 -9323.023,E2 -9323.023} C_VEL
LIN {X 0,Y 432.358,Z 158.628,A -85,B 0,C 180,E1 -9325.997,E2 -9325.997} C_VEL
LIN {X 0,Y 432.346,Z 158.629,A -85,B 0,C 180,E1 -9329.49,E2 -9329.49} C_VEL
LIN {X 0,Y 432.39,Z 158.626,A -85,B 0,C 180,E1 -9332.929,E2 -9332.929} C_VEL
LIN {X 0,Y 432.371,Z 158.627,A -85,B 0,C 180,E1 -9336.024,E2 -9336.024} C_VEL
LIN {X 0,Y 432.35,Z 158.63,A -85,B 0,C 180,E1 -9339.047,E2 -9339.047} C_VEL
LIN {X 0,Y 432.373,Z 158.628,A -85,B 0,C 180,E1 -9342.012,E2 -9342.012} C_VEL
LIN {X 0,Y 432.395,Z 158.624,A -85,B 0,C 180,E1 -9344.927,E2 -9344.927} C_VEL
LIN {X 0,Y 432.46,Z 158.617,A -85,B 0,C 180,E1 -9347.804,E2 -9347.804} C_VEL
LIN {X 0,Y 432.482,Z 158.613,A -85,B 0,C 180,E1 -9351.591,E2 -9351.591} C_VEL
LIN {X 0,Y 432.597,Z 158.601,A -85,B 0,C 180,E1 -9354.407,E2 -9354.407} C_VEL
LIN {X 0,Y 432.606,Z 158.601,A -85,B 0,C 180,E1 -9358.139,E2 -9358.139} C_VEL
LIN {X 0,Y 432.734,Z 158.584,A -85,B 0,C 180,E1 -9360,E2 -9360} C_VEL
LIN {X 0,Y 432.594,Z 158.599,A -85,B 0,C 180,E1 -9362.794,E2 -9362.794} C_VEL
LIN {X 0,Y 432.588,Z 158.603,A -85,B 0,C 180,E1 -9365.594,E2 -9365.594} C_VEL
LIN {X 0,Y 432.465,Z 158.616,A -85,B 0,C 180,E1 -9368.411,E2 -9368.411} C_VEL
LIN {X 0,Y 432.461,Z 158.618,A -85,B 0,C 180,E1 -9372.197,E2 -9372.197} C_VEL
LIN {X 0,Y 432.433,Z 158.622,A -85,B 0,C 180,E1 -9376.039,E2 -9376.039} C_VEL
LIN {X 0,Y 432.389,Z 158.627,A -85,B 0,C 180,E1 -9379.486,E2 -9379.486} C_VEL
LIN {X 0,Y 432.321,Z 158.633,A -85,B 0,C 180,E1 -9382.965,E2 -9382.965} C_VEL
LIN {X 0,Y 432.367,Z 158.627,A -85,B 0,C 180,E1 -9386.033,E2 -9386.033} C_VEL
LIN {X 0,Y 432.345,Z 158.632,A -85,B 0,C 180,E1 -9389.188,E2 -9389.188} C_VEL
LIN {X 0,Y 432.324,Z 158.632,A -85,B 0,C 180,E1 -9392.443,E2 -9392.443} C_VEL
LIN {X 0,Y 432.345,Z 158.631,A -85,B 0,C 180,E1 -9395.632,E2 -9395.632} C_VEL
LIN {X 0,Y 432.343,Z 158.631,A -85,B 0,C 180,E1 -9398.715,E2 -9398.715} C_VEL
LIN {X 0,Y 432.336,Z 158.631,A -85,B 0,C 180,E1 -9401.797,E2 -9401.797} C_VEL
LIN {X 0,Y 432.336,Z 158.628,A -85,B 0,C 180,E1 -9404.348,E2 -9404.348} C_VEL
LIN {X 0,Y 432.372,Z 158.797,A -85,B 0,C 180,E1 -9407.478,E2 -9407.478} C_VEL
LIN {X 0,Y 433.402,Z 164.289,A -85,B 0,C 180,E1 -9410.241,E2 -9410.241} C_VEL
LIN {X 0,Y 434.43,Z 170.573,A -85,B 0,C 180,E1 -9413.233,E2 -9413.233} C_VEL
LIN {X 0,Y 434.384,Z 174.45,A -85,B 0,C 180,E1 -9414.945,E2 -9414.945} C_VEL
LIN {X 0,Y 433.905,Z 182.223,A -85,B 0,C 180,E1 -9418.237,E2 -9418.237} C_VEL
LIN {X 0,Y 433.295,Z 191.353,A -85,B 0,C 180,E1 -9421.941,E2 -9421.941} C_VEL
LIN {X 0,Y 432.777,Z 200.268,A -85,B 0,C 180,E1 -9425.424,E2 -9425.424} C_VEL
LIN {X 0,Y 432.327,Z 209.822,A -85,B 0,C 180,E1 -9429.045,E2 -9429.045} C_VEL
LIN {X 0,Y 432.008,Z 217.821,A -85,B 0,C 180,E1 -9431.995,E2 -9431.995} C_VEL
LIN {X 0,Y 431.908,Z 221.385,A -85,B 0,C 180,E1 -9433.294,E2 -9433.294} C_VEL
LIN {X 0,Y 434.028,Z 234.855,A -85,B 0,C 180,E1 -9433.756,E2 -9433.756} C_VEL
LIN {X 0,Y 435.638,Z 245.443,A -85,B 0,C 180,E1 -9434.263,E2 -9434.263} C_VEL
LIN {X 0,Y 435.099,Z 257.102,A -85,B 0,C 180,E1 -9434.903,E2 -9434.903} C_VEL
LIN {X 0,Y 434.451,Z 268.484,A -85,B 0,C 180,E1 -9435.718,E2 -9435.718} C_VEL
LIN {X 0,Y 433.824,Z 279.39,A -85,B 0,C 180,E1 -9436.704,E2 -9436.704} C_VEL
LIN {X 0,Y 433.221,Z 289.421,A -85,B 0,C 180,E1 -9437.825,E2 -9437.825} C_VEL
LIN {X 0,Y 432.573,Z 297.953,A -85,B 0,C 180,E1 -9438.995,E2 -9438.995} C_VEL
LIN {X 0,Y 432.104,Z 306.286,A -85,B 0,C 180,E1 -9440.403,E2 -9440.403} C_VEL
LIN {X 0,Y 431.712,Z 313.004,A -85,B 0,C 180,E1 -9441.811,E2 -9441.811} C_VEL
LIN {X 0,Y 431.449,Z 319.162,A -85,B 0,C 180,E1 -9443.453,E2 -9443.453} C_VEL
LIN {X 0,Y 431.349,Z 323.164,A -85,B 0,C 180,E1 -9444.859,E2 -9444.859} C_VEL
LIN {X 0,Y 431.208,Z 326.114,A -85,B 0,C 180,E1 -9446.262,E2 -9446.262} C_VEL
LIN {X 0,Y 431.28,Z 327.526,A -85,B 0,C 180,E1 -9447.198,E2 -9447.198} C_VEL
LIN {X 0,Y 431.184,Z 329.131,A -85,B 0,C 180,E1 -9449.066,E2 -9449.066} C_VEL
LIN {X 0,Y 431.203,Z 329.345,A -85,B 0,C 180,E1 -9450,E2 -9450} C_VEL
LIN {X 0,Y 431.184,Z 329.119,A -85,B 0,C 180,E1 -9450.934,E2 -9450.934} C_VEL
LIN {X 0,Y 431.28,Z 327.489,A -85,B 0,C 180,E1 -9452.802,E2 -9452.802} C_VEL
LIN {X 0,Y 431.21,Z 326.062,A -85,B 0,C 180,E1 -9453.738,E2 -9453.738} C_VEL
LIN {X 0,Y 431.369,Z 323.088,A -85,B 0,C 180,E1 -9455.141,E2 -9455.141} C_VEL
LIN {X 0,Y 431.443,Z 319.055,A -85,B 0,C 180,E1 -9456.548,E2 -9456.548} C_VEL
LIN {X 0,Y 431.713,Z 312.869,A -85,B 0,C 180,E1 -9458.189,E2 -9458.189} C_VEL
LIN {X 0,Y 432.083,Z 306.115,A -85,B 0,C 180,E1 -9459.597,E2 -9459.597} C_VEL
LIN {X 0,Y 432.563,Z 297.744,A -85,B 0,C 180,E1 -9461.006,E2 -9461.006} C_VEL
LIN {X 0,Y 433.19,Z 289.178,A -85,B 0,C 180,E1 -9462.176,E2 -9462.176} C_VEL
LIN {X 0,Y 433.781,Z 279.29,A -85,B 0,C 180,E1 -9463.279,E2 -9463.279} C_VEL
LIN {X 0,Y 434.395,Z 268.161,A -85,B 0,C 180,E1 -9464.284,E2 -9464.284} C_VEL
LIN {X 0,Y 435.09,Z 256.749,A -85,B 0,C 180,E1 -9465.098,E2 -9465.098} C_VEL
LIN {X 0,Y 435.53,Z 245.043,A -85,B 0,C 180,E1 -9465.742,E2 -9465.742} C_VEL
LIN {X 0,Y 433.568,Z 231.847,A -85,B 0,C 180,E1 -9466.348,E2 -9466.348} C_VEL
LIN {X 0,Y 431.839,Z 220.798,A -85,B 0,C 180,E1 -9466.724,E2 -9466.724} C_VEL
LIN {X 0,Y 432.187,Z 211.862,A -85,B 0,C 180,E1 -9469.968,E2 -9469.968} C_VEL
LIN {X 0,Y 432.489,Z 203.819,A -85,B 0,C 180,E1 -9472.955,E2 -9472.955} C_VEL
LIN {X 0,Y 432.945,Z 194.819,A -85,B 0,C 180,E1 -9476.39,E2 -9476.39} C_VEL
LIN {X 0,Y 433.397,Z 186.66,A -85,B 0,C 180,E1 -9479.643,E2 -9479.643} C_VEL
LIN {X 0,Y 433.914,Z 179.536,A -85,B 0,C 180,E1 -9482.623,E2 -9482.623} C_VEL
LIN {X 0,Y 434.461,Z 172.711,A -85,B 0,C 180,E1 -9485.616,E2 -9485.616} C_VEL
LIN {X 0,Y 434.176,Z 168.731,A -85,B 0,C 180,E1 -9487.517,E2 -9487.517} C_VEL
LIN {X 0,Y 432.991,Z 161.995,A -85,B 0,C 180,E1 -9491.059,E2 -9491.059} C_VEL
LIN {X 0,Y 432.321,Z 158.63,A -85,B 0,C 180,E1 -9493.061,E2 -9493.061} C_VEL
LIN {X 0,Y 432.337,Z 158.634,A -85,B 0,C 180,E1 -9495.665,E2 -9495.665} C_VEL
LIN {X 0,Y 432.337,Z 158.636,A -85,B 0,C 180,E1 -9498.398,E2 -9498.398} C_VEL
LIN {X 0,Y 432.343,Z 158.635,A -85,B 0,C 180,E1 -9501.85,E2 -9501.85} C_VEL
LIN {X 0,Y 432.344,Z 158.632,A -85,B 0,C 180,E1 -9505.323,E2 -9505.323} C_VEL
LIN {X 0,Y 432.326,Z 158.634,A -85,B 0,C 180,E1 -9508.654,E2 -9508.654} C_VEL
LIN {X 0,Y 432.387,Z 158.627,A -85,B 0,C 180,E1 -9511.877,E2 -9511.877} C_VEL
LIN {X 0,Y 432.356,Z 158.63,A -85,B 0,C 180,E1 -9514.999,E2 -9514.999} C_VEL
LIN {X 0,Y 432.362,Z 158.629,A -85,B 0,C 180,E1 -9518.046,E2 -9518.046} C_VEL
LIN {X 0,Y 432.389,Z 158.627,A -85,B 0,C 180,E1 -9521.029,E2 -9521.029} C_VEL
LIN {X 0,Y 432.435,Z 158.62,A -85,B 0,C 180,E1 -9523.961,E2 -9523.961} C_VEL
LIN {X 0,Y 432.464,Z 158.618,A -85,B 0,C 180,E1 -9527.803,E2 -9527.803} C_VEL
LIN {X 0,Y 432.497,Z 158.614,A -85,B 0,C 180,E1 -9531.59,E2 -9531.59} C_VEL
LIN {X 0,Y 432.602,Z 158.6,A -85,B 0,C 180,E1 -9534.406,E2 -9534.406} C_VEL
LIN {X 0,Y 432.611,Z 158.599,A -85,B 0,C 180,E1 -9538.138,E2 -9538.138} C_VEL
LIN {X 0,Y 432.738,Z 158.584,A -85,B 0,C 180,E1 -9540,E2 -9540} C_VEL
LIN {X 0,Y 432.608,Z 158.6,A -85,B 0,C 180,E1 -9542.793,E2 -9542.793} C_VEL
LIN {X 0,Y 432.573,Z 158.607,A -85,B 0,C 180,E1 -9546.53,E2 -9546.53} C_VEL
LIN {X 0,Y 432.38,Z 158.629,A -85,B 0,C 180,E1 -9549.354,E2 -9549.354} C_VEL
LIN {X 0,Y 432.162,Z 158.726,A -85,B 0,C 180,E1 -9551.253,E2 -9551.253} C_VEL
LIN {X 0,Y 432.079,Z 161.478,A -85,B 0,C 180,E1 -9554.121,E2 -9554.121} C_VEL
LIN {X 0,Y 431.948,Z 164.306,A -85,B 0,C 180,E1 -9557.029,E2 -9557.029} C_VEL
LIN {X 0,Y 431.838,Z 167.26,A -85,B 0,C 180,E1 -9559.984,E2 -9559.984} C_VEL
LIN {X 0,Y 431.744,Z 170.269,A -85,B 0,C 180,E1 -9562.996,E2 -9562.996} C_VEL
LIN {X 0,Y 431.692,Z 173.392,A -85,B 0,C 180,E1 -9566.075,E2 -9566.075} C_VEL
LIN {X 0,Y 431.704,Z 175.978,A -85,B 0,C 180,E1 -9568.425,E2 -9568.425} C_VEL
LIN {X 0,Y 435.249,Z 189.649,A -85,B 0,C 180,E1 -9569.045,E2 -9569.045} C_VEL
LIN {X 0,Y 436.161,Z 193.719,A -85,B 0,C 180,E1 -9569.266,E2 -9569.266} C_VEL
LIN {X 0,Y 435.664,Z 206.28,A -85,B 0,C 180,E1 -9569.943,E2 -9569.943} C_VEL
LIN {X 0,Y 435.094,Z 217.237,A -85,B 0,C 180,E1 -9570.719,E2 -9570.719} C_VEL
LIN {X 0,Y 434.495,Z 228.281,A -85,B 0,C 180,E1 -9571.714,E2 -9571.714} C_VEL
LIN {X 0,Y 433.936,Z 237.786,A -85,B 0,C 180,E1 -9572.773,E2 -9572.773} C_VEL
LIN {X 0,Y 433.358,Z 246.749,A -85,B 0,C 180,E1 -9573.993,E2 -9573.993} C_VEL
LIN {X 0,Y 432.686,Z 255.091,A -85,B 0,C 180,E1 -9575.405,E2 -9575.405} C_VEL
LIN {X 0,Y 432.238,Z 262.465,A -85,B 0,C 180,E1 -9576.984,E2 -9576.984} C_VEL
LIN {X 0,Y 431.843,Z 268.361,A -85,B 0,C 180,E1 -9578.631,E2 -9578.631} C_VEL
LIN {X 0,Y 431.612,Z 272.222,A -85,B 0,C 180,E1 -9580.065,E2 -9580.065} C_VEL
LIN {X 0,Y 431.357,Z 275.644,A -85,B 0,C 180,E1 -9581.912,E2 -9581.912} C_VEL
LIN {X 0,Y 431.265,Z 277.033,A -85,B 0,C 180,E1 -9583.191,E2 -9583.191} C_VEL
LIN {X 0,Y 431.206,Z 277.693,A -85,B 0,C 180,E1 -9584.493,E2 -9584.493} C_VEL
LIN {X 0,Y 431.209,Z 277.582,A -85,B 0,C 180,E1 -9585.817,E2 -9585.817} C_VEL
LIN {X 0,Y 431.276,Z 276.621,A -85,B 0,C 180,E1 -9587.164,E2 -9587.164} C_VEL
LIN {X 0,Y 431.373,Z 274.768,A -85,B 0,C 180,E1 -9588.541,E2 -9588.541} C_VEL
LIN {X 0,Y 431.575,Z 271.949,A -85,B 0,C 180,E1 -9589.939,E2 -9589.939} C_VEL
LIN {X 0,Y 431.774,Z 267.994,A -85,B 0,C 180,E1 -9591.379,E2 -9591.379} C_VEL
LIN {X 0,Y 432.13,Z 262.094,A -85,B 0,C 180,E1 -9593.004,E2 -9593.004} C_VEL
LIN {X 0,Y 432.578,Z 254.539,A -85,B 0,C 180,E1 -9594.599,E2 -9594.599} C_VEL
LIN {X 0,Y 433.154,Z 245.983,A -85,B 0,C 180,E1 -9596.032,E2 -9596.032} C_VEL
LIN {X 0,Y 433.722,Z 236.915,A -85,B 0,C 180,E1 -9597.25,E2 -9597.25} C_VEL
LIN {X 0,Y 434.325,Z 226.304,A -85,B 0,C 180,E1 -9598.407,E2 -9598.407} C_VEL
LIN {X 0,Y 434.91,Z 214.85,A -85,B 0,C 180,E1 -9599.401,E2 -9599.401} C_VEL
LIN {X 0,Y 435.497,Z 202.798,A -85,B 0,C 180,E1 -9600.211,E2 -9600.211} C_VEL
LIN {X 0,Y 435.906,Z 193.725,A -85,B 0,C 180,E1 -9600.688,E2 -9600.688} C_VEL
LIN {X 0,Y 433.3,Z 181.648,A -85,B 0,C 180,E1 -9601.28,E2 -9601.28} C_VEL
LIN {X 0,Y 431.533,Z 174.332,A -85,B 0,C 180,E1 -9601.575,E2 -9601.575} C_VEL
LIN {X 0,Y 431.591,Z 170.637,A -85,B 0,C 180,E1 -9604.951,E2 -9604.951} C_VEL
LIN {X 0,Y 431.564,Z 167.188,A -85,B 0,C 180,E1 -9608.161,E2 -9608.161} C_VEL
LIN {X 0,Y 431.695,Z 164.159,A -85,B 0,C 180,E1 -9610.998,E2 -9610.998} C_VEL
LIN {X 0,Y 431.801,Z 161.076,A -85,B 0,C 180,E1 -9613.937,E2 -9613.937} C_VEL
LIN {X 0,Y 431.811,Z 159.077,A -85,B 0,C 180,E1 -9615.869,E2 -9615.869} C_VEL
LIN {X 0,Y 432.089,Z 158.665,A -85,B 0,C 180,E1 -9617.793,E2 -9617.793} C_VEL
LIN {X 0,Y 432.394,Z 158.623,A -85,B 0,C 180,E1 -9620.914,E2 -9620.914} C_VEL
LIN {X 0,Y 431.789,Z 158.701,A -85,B 0,C 180,E1 -9621.692,E2 -9621.692} C_VEL
LIN {X 0,Y 429.019,Z 159.044,A -85,B 0,C 180,E1 -9622.958,E2 -9622.958} C_VEL
LIN {X 0,Y 426.607,Z 159.348,A -85,B 0,C 180,E1 -9623.979,E2 -9623.979} C_VEL
LIN {X 0,Y 425.515,Z 159.482,A -85,B 0,C 180,E1 -9624.767,E2 -9624.767} C_VEL
LIN {X 0,Y 425.397,Z 159.495,A -85,B 0,C 180,E1 -9625.035,E2 -9625.035} C_VEL
LIN {X 0,Y 425.573,Z 159.476,A -85,B 0,C 180,E1 -9628.107,E2 -9628.107} C_VEL
LIN {X 0,Y 425.7,Z 159.461,A -85,B 0,C 180,E1 -9630,E2 -9630} C_VEL
LIN {X 0,Y 425.554,Z 159.475,A -85,B 0,C 180,E1 -9632.84,E2 -9632.84} C_VEL
LIN {X 0,Y 425.524,Z 159.48,A -85,B 0,C 180,E1 -9636.639,E2 -9636.639} C_VEL
LIN {X 0,Y 425.398,Z 159.497,A -85,B 0,C 180,E1 -9639.509,E2 -9639.509} C_VEL
LIN {X 0,Y 425.39,Z 159.495,A -85,B 0,C 180,E1 -9642.904,E2 -9642.904} C_VEL
LIN {X 0,Y 425.358,Z 159.5,A -85,B 0,C 180,E1 -9646.605,E2 -9646.605} C_VEL
LIN {X 0,Y 425.325,Z 159.507,A -85,B 0,C 180,E1 -9649.636,E2 -9649.636} C_VEL
LIN {X 0,Y 425.304,Z 159.51,A -85,B 0,C 180,E1 -9653.365,E2 -9653.365} C_VEL
LIN {X 0,Y 425.345,Z 159.503,A -85,B 0,C 180,E1 -9656.845,E2 -9656.845} C_VEL
LIN {X 0,Y 425.288,Z 159.512,A -85,B 0,C 180,E1 -9659.72,E2 -9659.72} C_VEL
LIN {X 0,Y 425.279,Z 159.512,A -85,B 0,C 180,E1 -9663.048,E2 -9663.048} C_VEL
LIN {X 0,Y 425.279,Z 159.511,A -85,B 0,C 180,E1 -9665.929,E2 -9665.929} C_VEL
LIN {X 0,Y 425.295,Z 159.511,A -85,B 0,C 180,E1 -9669.044,E2 -9669.044} C_VEL
LIN {X 0,Y 425.275,Z 159.513,A -85,B 0,C 180,E1 -9672.653,E2 -9672.653} C_VEL
LIN {X 0,Y 425.259,Z 159.512,A -85,B 0,C 180,E1 -9676.045,E2 -9676.045} C_VEL
LIN {X 0,Y 425.272,Z 159.514,A -85,B 0,C 180,E1 -9678.622,E2 -9678.622} C_VEL
LIN {X 0,Y 425.311,Z 159.508,A -85,B 0,C 180,E1 -9681.103,E2 -9681.103} C_VEL
LIN {X 0,Y 425.298,Z 159.51,A -85,B 0,C 180,E1 -9684.665,E2 -9684.665} C_VEL
LIN {X 0,Y 425.263,Z 159.513,A -85,B 0,C 180,E1 -9688.074,E2 -9688.074} C_VEL
LIN {X 0,Y 425.33,Z 159.504,A -85,B 0,C 180,E1 -9691.368,E2 -9691.368} C_VEL
LIN {X 0,Y 425.295,Z 159.51,A -85,B 0,C 180,E1 -9694.555,E2 -9694.555} C_VEL
LIN {X 0,Y 425.287,Z 159.509,A -85,B 0,C 180,E1 -9697.662,E2 -9697.662} C_VEL
LIN {X 0,Y 425.361,Z 159.502,A -85,B 0,C 180,E1 -9700.705,E2 -9700.705} C_VEL
LIN {X 0,Y 425.388,Z 159.497,A -85,B 0,C 180,E1 -9703.689,E2 -9703.689} C_VEL
LIN {X 0,Y 425.413,Z 159.494,A -85,B 0,C 180,E1 -9707.599,E2 -9707.599} C_VEL
LIN {X 0,Y 425.436,Z 159.49,A -85,B 0,C 180,E1 -9711.45,E2 -9711.45} C_VEL
LIN {X 0,Y 425.553,Z 159.48,A -85,B 0,C 180,E1 -9714.314,E2 -9714.314} C_VEL
LIN {X 0,Y 425.576,Z 159.477,A -85,B 0,C 180,E1 -9718.108,E2 -9718.108} C_VEL
LIN {X 0,Y 425.703,Z 159.46,A -85,B 0,C 180,E1 -9720,E2 -9720} C_VEL
LIN {X 0,Y 425.547,Z 159.477,A -85,B 0,C 180,E1 -9722.84,E2 -9722.84} C_VEL
LIN {X 0,Y 425.544,Z 159.48,A -85,B 0,C 180,E1 -9725.687,E2 -9725.687} C_VEL
LIN {X 0,Y 425.41,Z 159.494,A -85,B 0,C 180,E1 -9728.551,E2 -9728.551} C_VEL
LIN {X 0,Y 425.414,Z 159.494,A -85,B 0,C 180,E1 -9732.402,E2 -9732.402} C_VEL
LIN {X 0,Y 425.391,Z 159.496,A -85,B 0,C 180,E1 -9736.312,E2 -9736.312} C_VEL
LIN {X 0,Y 425.331,Z 159.507,A -85,B 0,C 180,E1 -9739.636,E2 -9739.636} C_VEL
LIN {X 0,Y 425.309,Z 159.509,A -85,B 0,C 180,E1 -9743.365,E2 -9743.365} C_VEL
LIN {X 0,Y 425.35,Z 159.501,A -85,B 0,C 180,E1 -9746.844,E2 -9746.844} C_VEL
LIN {X 0,Y 425.293,Z 159.51,A -85,B 0,C 180,E1 -9749.72,E2 -9749.72} C_VEL
LIN {X 0,Y 425.284,Z 159.512,A -85,B 0,C 180,E1 -9753.048,E2 -9753.048} C_VEL
LIN {X 0,Y 425.283,Z 159.509,A -85,B 0,C 180,E1 -9755.929,E2 -9755.929} C_VEL
LIN {X 0,Y 425.29,Z 159.511,A -85,B 0,C 180,E1 -9759.042,E2 -9759.042} C_VEL
LIN {X 0,Y 425.292,Z 159.508,A -85,B 0,C 180,E1 -9761.958,E2 -9761.958} C_VEL
LIN {X 0,Y 425.287,Z 159.506,A -85,B 0,C 180,E1 -9765.283,E2 -9765.283} C_VEL
LIN {X 0,Y 425.319,Z 159.681,A -85,B 0,C 180,E1 -9767.144,E2 -9767.144} C_VEL
LIN {X 0,Y 426.368,Z 165.226,A -85,B 0,C 180,E1 -9769.995,E2 -9769.995} C_VEL
LIN {X 0,Y 427.418,Z 171.677,A -85,B 0,C 180,E1 -9773.119,E2 -9773.119} C_VEL
LIN {X 0,Y 427.413,Z 175.529,A -85,B 0,C 180,E1 -9774.865,E2 -9774.865} C_VEL
LIN {X 0,Y 426.899,Z 183.304,A -85,B 0,C 180,E1 -9778.21,E2 -9778.21} C_VEL
LIN {X 0,Y 426.252,Z 192.422,A -85,B 0,C 180,E1 -9781.972,E2 -9781.972} C_VEL
LIN {X 0,Y 425.733,Z 200.571,A -85,B 0,C 180,E1 -9785.223,E2 -9785.223} C_VEL
LIN {X 0,Y 425.285,Z 209.521,A -85,B 0,C 180,E1 -9788.681,E2 -9788.681} C_VEL
LIN {X 0,Y 424.949,Z 217.426,A -85,B 0,C 180,E1 -9791.686,E2 -9791.686} C_VEL
LIN {X 0,Y 424.837,Z 220.919,A -85,B 0,C 180,E1 -9792.99,E2 -9792.99} C_VEL
LIN {X 0,Y 427.204,Z 236.007,A -85,B 0,C 180,E1 -9793.549,E2 -9793.549} C_VEL
LIN {X 0,Y 428.69,Z 247.386,A -85,B 0,C 180,E1 -9794.123,E2 -9794.123} C_VEL
LIN {X 0,Y 427.974,Z 260.207,A -85,B 0,C 180,E1 -9794.889,E2 -9794.889} C_VEL
LIN {X 0,Y 427.33,Z 270.911,A -85,B 0,C 180,E1 -9795.718,E2 -9795.718} C_VEL
LIN {X 0,Y 426.674,Z 281.873,A -85,B 0,C 180,E1 -9796.789,E2 -9796.789} C_VEL
LIN {X 0,Y 426.105,Z 290.814,A -85,B 0,C 180,E1 -9797.861,E2 -9797.861} C_VEL
LIN {X 0,Y 425.385,Z 300.528,A -85,B 0,C 180,E1 -9799.288,E2 -9799.288} C_VEL
LIN {X 0,Y 424.903,Z 308.284,A -85,B 0,C 180,E1 -9800.72,E2 -9800.72} C_VEL
LIN {X 0,Y 424.466,Z 315.425,A -85,B 0,C 180,E1 -9802.388,E2 -9802.388} C_VEL
LIN {X 0,Y 424.276,Z 320.571,A -85,B 0,C 180,E1 -9803.947,E2 -9803.947} C_VEL
LIN {X 0,Y 424.224,Z 323.827,A -85,B 0,C 180,E1 -9805.249,E2 -9805.249} C_VEL
LIN {X 0,Y 424.119,Z 325.699,A -85,B 0,C 180,E1 -9806.2,E2 -9806.2} C_VEL
LIN {X 0,Y 424.192,Z 327.112,A -85,B 0,C 180,E1 -9807.151,E2 -9807.151} C_VEL
LIN {X 0,Y 424.103,Z 328.715,A -85,B 0,C 180,E1 -9809.051,E2 -9809.051} C_VEL
LIN {X 0,Y 424.118,Z 328.927,A -85,B 0,C 180,E1 -9810,E2 -9810} C_VEL
LIN {X 0,Y 424.103,Z 328.7,A -85,B 0,C 180,E1 -9810.95,E2 -9810.95} C_VEL
LIN {X 0,Y 424.192,Z 327.063,A -85,B 0,C 180,E1 -9812.849,E2 -9812.849} C_VEL
LIN {X 0,Y 424.121,Z 325.634,A -85,B 0,C 180,E1 -9813.801,E2 -9813.801} C_VEL
LIN {X 0,Y 424.28,Z 322.654,A -85,B 0,C 180,E1 -9815.227,E2 -9815.227} C_VEL
LIN {X 0,Y 424.361,Z 318.615,A -85,B 0,C 180,E1 -9816.657,E2 -9816.657} C_VEL
LIN {X 0,Y 424.652,Z 312.42,A -85,B 0,C 180,E1 -9818.327,E2 -9818.327} C_VEL
LIN {X 0,Y 425.031,Z 305.659,A -85,B 0,C 180,E1 -9819.758,E2 -9819.758} C_VEL
LIN {X 0,Y 425.557,Z 297.283,A -85,B 0,C 180,E1 -9821.189,E2 -9821.189} C_VEL
LIN {X 0,Y 426.203,Z 288.709,A -85,B 0,C 180,E1 -9822.379,E2 -9822.379} C_VEL
LIN {X 0,Y 426.847,Z 278.17,A -85,B 0,C 180,E1 -9823.565,E2 -9823.565} C_VEL
LIN {X 0,Y 427.547,Z 266.247,A -85,B 0,C 180,E1 -9824.64,E2 -9824.64} C_VEL
LIN {X 0,Y 428.327,Z 254.329,A -85,B 0,C 180,E1 -9825.464,E2 -9825.464} C_VEL
LIN {X 0,Y 428.601,Z 245.806,A -85,B 0,C 180,E1 -9825.942,E2 -9825.942} C_VEL
LIN {X 0,Y 426.621,Z 232.13,A -85,B 0,C 180,E1 -9826.598,E2 -9826.598} C_VEL
LIN {X 0,Y 424.773,Z 220.361,A -85,B 0,C 180,E1 -9827.009,E2 -9827.009} C_VEL
LIN {X 0,Y 425.109,Z 212.638,A -85,B 0,C 180,E1 -9829.874,E2 -9829.874} C_VEL
LIN {X 0,Y 425.459,Z 203.464,A -85,B 0,C 180,E1 -9833.357,E2 -9833.357} C_VEL
LIN {X 0,Y 425.907,Z 195.504,A -85,B 0,C 180,E1 -9836.458,E2 -9836.458} C_VEL
LIN {X 0,Y 426.371,Z 187.668,A -85,B 0,C 180,E1 -9839.637,E2 -9839.637} C_VEL
LIN {X 0,Y 426.943,Z 180.023,A -85,B 0,C 180,E1 -9842.91,E2 -9842.91} C_VEL
LIN {X 0,Y 427.495,Z 173.851,A -85,B 0,C 180,E1 -9845.706,E2 -9845.706} C_VEL
LIN {X 0,Y 427.109,Z 169.522,A -85,B 0,C 180,E1 -9847.83,E2 -9847.83} C_VEL
LIN {X 0,Y 425.98,Z 163.123,A -85,B 0,C 180,E1 -9851.295,E2 -9851.295} C_VEL
LIN {X 0,Y 425.273,Z 159.509,A -85,B 0,C 180,E1 -9853.486,E2 -9853.486} C_VEL
LIN {X 0,Y 425.262,Z 159.517,A -85,B 0,C 180,E1 -9856.649,E2 -9856.649} C_VEL
LIN {X 0,Y 425.299,Z 159.513,A -85,B 0,C 180,E1 -9859.874,E2 -9859.874} C_VEL
LIN {X 0,Y 425.283,Z 159.513,A -85,B 0,C 180,E1 -9862.488,E2 -9862.488} C_VEL
LIN {X 0,Y 425.312,Z 159.507,A -85,B 0,C 180,E1 -9865.817,E2 -9865.817} C_VEL
LIN {X 0,Y 425.295,Z 159.509,A -85,B 0,C 180,E1 -9869.239,E2 -9869.239} C_VEL
LIN {X 0,Y 425.354,Z 159.503,A -85,B 0,C 180,E1 -9872.442,E2 -9872.442} C_VEL
LIN {X 0,Y 425.356,Z 159.502,A -85,B 0,C 180,E1 -9875.602,E2 -9875.602} C_VEL
LIN {X 0,Y 425.298,Z 159.51,A -85,B 0,C 180,E1 -9878.681,E2 -9878.681} C_VEL
LIN {X 0,Y 425.326,Z 159.504,A -85,B 0,C 180,E1 -9881.702,E2 -9881.702} C_VEL
LIN {X 0,Y 425.353,Z 159.503,A -85,B 0,C 180,E1 -9884.67,E2 -9884.67} C_VEL
LIN {X 0,Y 425.417,Z 159.496,A -85,B 0,C 180,E1 -9887.598,E2 -9887.598} C_VEL
LIN {X 0,Y 425.447,Z 159.492,A -85,B 0,C 180,E1 -9891.45,E2 -9891.45} C_VEL
LIN {X 0,Y 425.559,Z 159.477,A -85,B 0,C 180,E1 -9894.313,E2 -9894.313} C_VEL
LIN {X 0,Y 425.58,Z 159.475,A -85,B 0,C 180,E1 -9898.107,E2 -9898.107} C_VEL
LIN {X 0,Y 425.708,Z 159.46,A -85,B 0,C 180,E1 -9900,E2 -9900} C_VEL
LIN {X 0,Y 425.56,Z 159.479,A -85,B 0,C 180,E1 -9902.839,E2 -9902.839} C_VEL
LIN {X 0,Y 425.531,Z 159.485,A -85,B 0,C 180,E1 -9906.638,E2 -9906.638} C_VEL
LIN {X 0,Y 425.33,Z 159.507,A -85,B 0,C 180,E1 -9909.51,E2 -9909.51} C_VEL
LIN {X 0,Y 425.127,Z 159.874,A -85,B 0,C 180,E1 -9911.442,E2 -9911.442} C_VEL
LIN {X 0,Y 425.031,Z 162.686,A -85,B 0,C 180,E1 -9914.36,E2 -9914.36} C_VEL
LIN {X 0,Y 424.908,Z 165.512,A -85,B 0,C 180,E1 -9917.32,E2 -9917.32} C_VEL
LIN {X 0,Y 424.786,Z 168.465,A -85,B 0,C 180,E1 -9920.33,E2 -9920.33} C_VEL
LIN {X 0,Y 424.695,Z 171.502,A -85,B 0,C 180,E1 -9923.4,E2 -9923.4} C_VEL
LIN {X 0,Y 424.617,Z 174.764,A -85,B 0,C 180,E1 -9926.648,E2 -9926.648} C_VEL
LIN {X 0,Y 424.614,Z 176.255,A -85,B 0,C 180,E1 -9928.112,E2 -9928.112} C_VEL
LIN {X 0,Y 428.314,Z 190.389,A -85,B 0,C 180,E1 -9928.78,E2 -9928.78} C_VEL
LIN {X 0,Y 429.335,Z 195.829,A -85,B 0,C 180,E1 -9929.08,E2 -9929.08} C_VEL
LIN {X 0,Y 428.843,Z 206.979,A -85,B 0,C 180,E1 -9929.705,E2 -9929.705} C_VEL
LIN {X 0,Y 428.192,Z 218.938,A -85,B 0,C 180,E1 -9930.584,E2 -9930.584} C_VEL
LIN {X 0,Y 427.565,Z 229.872,A -85,B 0,C 180,E1 -9931.606,E2 -9931.606} C_VEL
LIN {X 0,Y 426.87,Z 240.116,A -85,B 0,C 180,E1 -9932.8,E2 -9932.8} C_VEL
LIN {X 0,Y 426.246,Z 249.038,A -85,B 0,C 180,E1 -9934.096,E2 -9934.096} C_VEL
LIN {X 0,Y 425.536,Z 257.56,A -85,B 0,C 180,E1 -9935.633,E2 -9935.633} C_VEL
LIN {X 0,Y 425.178,Z 263.516,A -85,B 0,C 180,E1 -9936.99,E2 -9936.99} C_VEL
LIN {X 0,Y 424.859,Z 268.259,A -85,B 0,C 180,E1 -9938.333,E2 -9938.333} C_VEL
LIN {X 0,Y 424.535,Z 273.185,A -85,B 0,C 180,E1 -9940.212,E2 -9940.212} C_VEL
LIN {X 0,Y 424.284,Z 276.016,A -85,B 0,C 180,E1 -9941.806,E2 -9941.806} C_VEL
LIN {X 0,Y 424.179,Z 277.504,A -85,B 0,C 180,E1 -9943.196,E2 -9943.196} C_VEL
LIN {X 0,Y 424.116,Z 278.135,A -85,B 0,C 180,E1 -9944.557,E2 -9944.557} C_VEL
LIN {X 0,Y 424.122,Z 277.973,A -85,B 0,C 180,E1 -9945.895,E2 -9945.895} C_VEL
LIN {X 0,Y 424.192,Z 277.029,A -85,B 0,C 180,E1 -9947.212,E2 -9947.212} C_VEL
LIN {X 0,Y 424.283,Z 275.326,A -85,B 0,C 180,E1 -9948.503,E2 -9948.503} C_VEL
LIN {X 0,Y 424.486,Z 272.888,A -85,B 0,C 180,E1 -9949.781,E2 -9949.781} C_VEL
LIN {X 0,Y 424.658,Z 269.651,A -85,B 0,C 180,E1 -9951.062,E2 -9951.062} C_VEL
LIN {X 0,Y 424.971,Z 264.768,A -85,B 0,C 180,E1 -9952.542,E2 -9952.542} C_VEL
LIN {X 0,Y 425.345,Z 258.371,A -85,B 0,C 180,E1 -9954.059,E2 -9954.059} C_VEL
LIN {X 0,Y 425.818,Z 251.175,A -85,B 0,C 180,E1 -9955.427,E2 -9955.427} C_VEL
LIN {X 0,Y 426.489,Z 242.4,A -85,B 0,C 180,E1 -9956.775,E2 -9956.775} C_VEL
LIN {X 0,Y 427.033,Z 233.037,A -85,B 0,C 180,E1 -9957.943,E2 -9957.943} C_VEL
LIN {X 0,Y 427.667,Z 222.081,A -85,B 0,C 180,E1 -9959.048,E2 -9959.048} C_VEL
LIN {X 0,Y 428.215,Z 211.352,A -85,B 0,C 180,E1 -9959.914,E2 -9959.914} C_VEL
LIN {X 0,Y 428.883,Z 199.199,A -85,B 0,C 180,E1 -9960.669,E2 -9960.669} C_VEL
LIN {X 0,Y 428.958,Z 194.102,A -85,B 0,C 180,E1 -9960.933,E2 -9960.933} C_VEL
LIN {X 0,Y 425.895,Z 180.576,A -85,B 0,C 180,E1 -9961.604,E2 -9961.604} C_VEL
LIN {X 0,Y 424.485,Z 174.709,A -85,B 0,C 180,E1 -9961.845,E2 -9961.845} C_VEL
LIN {X 0,Y 424.518,Z 171.813,A -85,B 0,C 180,E1 -9964.505,E2 -9964.505} C_VEL
LIN {X 0,Y 424.51,Z 168.09,A -85,B 0,C 180,E1 -9967.987,E2 -9967.987} C_VEL
LIN {X 0,Y 424.62,Z 165.248,A -85,B 0,C 180,E1 -9970.669,E2 -9970.669} C_VEL
LIN {X 0,Y 424.731,Z 162.124,A -85,B 0,C 180,E1 -9973.681,E2 -9973.681} C_VEL
LIN {X 0,Y 424.741,Z 160.103,A -85,B 0,C 180,E1 -9975.629,E2 -9975.629} C_VEL
LIN {X 0,Y 424.839,Z 159.57,A -85,B 0,C 180,E1 -9976.609,E2 -9976.609} C_VEL
LIN {X 0,Y 425.219,Z 159.518,A -85,B 0,C 180,E1 -9979.525,E2 -9979.525} C_VEL
LIN {X 0,Y 425.495,Z 159.486,A -85,B 0,C 180,E1 -9982.407,E2 -9982.407} C_VEL
LIN {X 0,Y 425.543,Z 159.479,A -85,B 0,C 180,E1 -9984.313,E2 -9984.313} C_VEL
LIN {X 0,Y 425.397,Z 159.495,A -85,B 0,C 180,E1 -9985.035,E2 -9985.035} C_VEL
LIN {X 0,Y 424.654,Z 159.59,A -85,B 0,C 180,E1 -9985.826,E2 -9985.826} C_VEL
LIN {X 0,Y 421.808,Z 159.944,A -85,B 0,C 180,E1 -9987.112,E2 -9987.112} C_VEL
LIN {X 0,Y 419.493,Z 160.233,A -85,B 0,C 180,E1 -9988.151,E2 -9988.151} C_VEL
LIN {X 0,Y 418.566,Z 160.346,A -85,B 0,C 180,E1 -9988.953,E2 -9988.953} C_VEL
LIN {X 0,Y 418.522,Z 160.351,A -85,B 0,C 180,E1 -9989.224,E2 -9989.224} C_VEL
LIN {X 0,Y 418.67,Z 160.337,A -85,B 0,C 180,E1 -9990,E2 -9990} C_VEL
LIN {X 0,Y 418.507,Z 160.352,A -85,B 0,C 180,E1 -9992.888,E2 -9992.888} C_VEL
LIN {X 0,Y 418.488,Z 160.356,A -85,B 0,C 180,E1 -9996.751,E2 -9996.751} C_VEL
LIN {X 0,Y 418.397,Z 160.367,A -85,B 0,C 180,E1 -9998.695,E2 -9998.695} C_VEL
LIN {X 0,Y 418.312,Z 160.38,A -85,B 0,C 180,E1 -10001.631,E2 -10001.631} C_VEL
LIN {X 0,Y 418.3,Z 160.379,A -85,B 0,C 180,E1 -10004.597,E2 -10004.597} C_VEL
LIN {X 0,Y 418.285,Z 160.384,A -85,B 0,C 180,E1 -10007.604,E2 -10007.604} C_VEL
LIN {X 0,Y 418.247,Z 160.386,A -85,B 0,C 180,E1 -10010.663,E2 -10010.663} C_VEL
LIN {X 0,Y 418.285,Z 160.384,A -85,B 0,C 180,E1 -10013.781,E2 -10013.781} C_VEL
LIN {X 0,Y 418.307,Z 160.381,A -85,B 0,C 180,E1 -10017.071,E2 -10017.071} C_VEL
LIN {X 0,Y 418.241,Z 160.386,A -85,B 0,C 180,E1 -10020.272,E2 -10020.272} C_VEL
LIN {X 0,Y 418.245,Z 160.388,A -85,B 0,C 180,E1 -10023.677,E2 -10023.677} C_VEL
LIN {X 0,Y 418.237,Z 160.39,A -85,B 0,C 180,E1 -10027.224,E2 -10027.224} C_VEL
LIN {X 0,Y 418.248,Z 160.387,A -85,B 0,C 180,E1 -10029.682,E2 -10029.682} C_VEL
LIN {X 0,Y 418.229,Z 160.388,A -85,B 0,C 180,E1 -10032.322,E2 -10032.322} C_VEL
LIN {X 0,Y 418.235,Z 160.39,A -85,B 0,C 180,E1 -10035.109,E2 -10035.109} C_VEL
LIN {X 0,Y 418.238,Z 160.387,A -85,B 0,C 180,E1 -10037.767,E2 -10037.767} C_VEL
LIN {X 0,Y 418.255,Z 160.387,A -85,B 0,C 180,E1 -10040.619,E2 -10040.619} C_VEL
LIN {X 0,Y 418.244,Z 160.386,A -85,B 0,C 180,E1 -10043.977,E2 -10043.977} C_VEL
LIN {X 0,Y 418.256,Z 160.386,A -85,B 0,C 180,E1 -10047.157,E2 -10047.157} C_VEL
LIN {X 0,Y 418.267,Z 160.386,A -85,B 0,C 180,E1 -10050.896,E2 -10050.896} C_VEL
LIN {X 0,Y 418.27,Z 160.384,A -85,B 0,C 180,E1 -10054.097,E2 -10054.097} C_VEL
LIN {X 0,Y 418.238,Z 160.388,A -85,B 0,C 180,E1 -10057.264,E2 -10057.264} C_VEL
LIN {X 0,Y 418.283,Z 160.384,A -85,B 0,C 180,E1 -10060.365,E2 -10060.365} C_VEL
LIN {X 0,Y 418.316,Z 160.377,A -85,B 0,C 180,E1 -10063.405,E2 -10063.405} C_VEL
LIN {X 0,Y 418.347,Z 160.374,A -85,B 0,C 180,E1 -10067,E2 -10067} C_VEL
LIN {X 0,Y 418.341,Z 160.377,A -85,B 0,C 180,E1 -10070.329,E2 -10070.329} C_VEL
LIN {X 0,Y 418.48,Z 160.357,A -85,B 0,C 180,E1 -10073.249,E2 -10073.249} C_VEL
LIN {X 0,Y 418.341,Z 160.373,A -85,B 0,C 180,E1 -10075.182,E2 -10075.182} C_VEL
LIN {X 0,Y 418.546,Z 160.352,A -85,B 0,C 180,E1 -10078.076,E2 -10078.076} C_VEL
LIN {X 0,Y 418.673,Z 160.335,A -85,B 0,C 180,E1 -10080,E2 -10080} C_VEL
LIN {X 0,Y 418.502,Z 160.354,A -85,B 0,C 180,E1 -10082.888,E2 -10082.888} C_VEL
LIN {X 0,Y 418.501,Z 160.357,A -85,B 0,C 180,E1 -10085.783,E2 -10085.783} C_VEL
LIN {X 0,Y 418.379,Z 160.369,A -85,B 0,C 180,E1 -10088.696,E2 -10088.696} C_VEL
LIN {X 0,Y 418.317,Z 160.381,A -85,B 0,C 180,E1 -10091.631,E2 -10091.631} C_VEL
LIN {X 0,Y 418.305,Z 160.378,A -85,B 0,C 180,E1 -10094.597,E2 -10094.597} C_VEL
LIN {X 0,Y 418.29,Z 160.384,A -85,B 0,C 180,E1 -10097.604,E2 -10097.604} C_VEL
LIN {X 0,Y 418.252,Z 160.384,A -85,B 0,C 180,E1 -10100.663,E2 -10100.663} C_VEL
LIN {X 0,Y 418.29,Z 160.382,A -85,B 0,C 180,E1 -10103.781,E2 -10103.781} C_VEL
LIN {X 0,Y 418.312,Z 160.379,A -85,B 0,C 180,E1 -10107.071,E2 -10107.071} C_VEL
LIN {X 0,Y 418.247,Z 160.385,A -85,B 0,C 180,E1 -10110.272,E2 -10110.272} C_VEL
LIN {X 0,Y 418.249,Z 160.387,A -85,B 0,C 180,E1 -10113.678,E2 -10113.678} C_VEL
LIN {X 0,Y 418.242,Z 160.389,A -85,B 0,C 180,E1 -10117.224,E2 -10117.224} C_VEL
LIN {X 0,Y 418.249,Z 160.387,A -85,B 0,C 180,E1 -10119.683,E2 -10119.683} C_VEL
LIN {X 0,Y 418.232,Z 160.387,A -85,B 0,C 180,E1 -10122.321,E2 -10122.321} C_VEL
LIN {X 0,Y 418.238,Z 160.384,A -85,B 0,C 180,E1 -10125.109,E2 -10125.109} C_VEL
LIN {X 0,Y 418.261,Z 160.493,A -85,B 0,C 180,E1 -10126.77,E2 -10126.77} C_VEL
LIN {X 0,Y 419.346,Z 166.293,A -85,B 0,C 180,E1 -10129.817,E2 -10129.817} C_VEL
LIN {X 0,Y 420.244,Z 171.55,A -85,B 0,C 180,E1 -10132.429,E2 -10132.429} C_VEL
LIN {X 0,Y 420.524,Z 175.318,A -85,B 0,C 180,E1 -10134.202,E2 -10134.202} C_VEL
LIN {X 0,Y 419.973,Z 183.065,A -85,B 0,C 180,E1 -10137.622,E2 -10137.622} C_VEL
LIN {X 0,Y 419.335,Z 190.84,A -85,B 0,C 180,E1 -10140.92,E2 -10140.92} C_VEL
LIN {X 0,Y 418.863,Z 198.684,A -85,B 0,C 180,E1 -10144.135,E2 -10144.135} C_VEL
LIN {X 0,Y 418.389,Z 207.12,A -85,B 0,C 180,E1 -10147.5,E2 -10147.5} C_VEL
LIN {X 0,Y 418,Z 215.764,A -85,B 0,C 180,E1 -10150.861,E2 -10150.861} C_VEL
LIN {X 0,Y 417.792,Z 220.815,A -85,B 0,C 180,E1 -10152.718,E2 -10152.718} C_VEL
LIN {X 0,Y 420.006,Z 234.474,A -85,B 0,C 180,E1 -10153.215,E2 -10153.215} C_VEL
LIN {X 0,Y 421.804,Z 246.965,A -85,B 0,C 180,E1 -10153.857,E2 -10153.857} C_VEL
LIN {X 0,Y 421.246,Z 258.032,A -85,B 0,C 180,E1 -10154.518,E2 -10154.518} C_VEL
LIN {X 0,Y 420.54,Z 269.067,A -85,B 0,C 180,E1 -10155.359,E2 -10155.359} C_VEL
LIN {X 0,Y 419.906,Z 278.72,A -85,B 0,C 180,E1 -10156.273,E2 -10156.273} C_VEL
LIN {X 0,Y 419.244,Z 288.579,A -85,B 0,C 180,E1 -10157.413,E2 -10157.413} C_VEL
LIN {X 0,Y 418.574,Z 297.118,A -85,B 0,C 180,E1 -10158.622,E2 -10158.622} C_VEL
LIN {X 0,Y 418.017,Z 305.449,A -85,B 0,C 180,E1 -10160.077,E2 -10160.077} C_VEL
LIN {X 0,Y 417.589,Z 312.17,A -85,B 0,C 180,E1 -10161.532,E2 -10161.532} C_VEL
LIN {X 0,Y 417.272,Z 318.331,A -85,B 0,C 180,E1 -10163.229,E2 -10163.229} C_VEL
LIN {X 0,Y 417.181,Z 322.335,A -85,B 0,C 180,E1 -10164.684,E2 -10164.684} C_VEL
LIN {X 0,Y 417.034,Z 325.284,A -85,B 0,C 180,E1 -10166.135,E2 -10166.135} C_VEL
LIN {X 0,Y 417.092,Z 326.696,A -85,B 0,C 180,E1 -10167.103,E2 -10167.103} C_VEL
LIN {X 0,Y 417.058,Z 327.694,A -85,B 0,C 180,E1 -10168.069,E2 -10168.069} C_VEL
LIN {X 0,Y 417.036,Z 328.509,A -85,B 0,C 180,E1 -10170,E2 -10170} C_VEL
LIN {X 0,Y 417.024,Z 328.281,A -85,B 0,C 180,E1 -10170.966,E2 -10170.966} C_VEL
LIN {X 0,Y 417.058,Z 327.656,A -85,B 0,C 180,E1 -10171.932,E2 -10171.932} C_VEL
LIN {X 0,Y 417.107,Z 326.637,A -85,B 0,C 180,E1 -10172.898,E2 -10172.898} C_VEL
LIN {X 0,Y 417.036,Z 325.205,A -85,B 0,C 180,E1 -10173.865,E2 -10173.865} C_VEL
LIN {X 0,Y 417.193,Z 322.22,A -85,B 0,C 180,E1 -10175.316,E2 -10175.316} C_VEL
LIN {X 0,Y 417.277,Z 318.175,A -85,B 0,C 180,E1 -10176.771,E2 -10176.771} C_VEL
LIN {X 0,Y 417.59,Z 311.971,A -85,B 0,C 180,E1 -10178.468,E2 -10178.468} C_VEL
LIN {X 0,Y 418.004,Z 305.204,A -85,B 0,C 180,E1 -10179.924,E2 -10179.924} C_VEL
LIN {X 0,Y 418.565,Z 296.824,A -85,B 0,C 180,E1 -10181.379,E2 -10181.379} C_VEL
LIN {X 0,Y 419.21,Z 288.245,A -85,B 0,C 180,E1 -10182.588,E2 -10182.588} C_VEL
LIN {X 0,Y 419.893,Z 277.514,A -85,B 0,C 180,E1 -10183.814,E2 -10183.814} C_VEL
LIN {X 0,Y 420.656,Z 265.792,A -85,B 0,C 180,E1 -10184.885,E2 -10184.885} C_VEL
LIN {X 0,Y 421.474,Z 253.886,A -85,B 0,C 180,E1 -10185.722,E2 -10185.722} C_VEL
LIN {X 0,Y 421.679,Z 246.496,A -85,B 0,C 180,E1 -10186.149,E2 -10186.149} C_VEL
LIN {X 0,Y 419.753,Z 232.891,A -85,B 0,C 180,E1 -10186.838,E2 -10186.838} C_VEL
LIN {X 0,Y 417.72,Z 219.904,A -85,B 0,C 180,E1 -10187.316,E2 -10187.316} C_VEL
LIN {X 0,Y 418.05,Z 212.409,A -85,B 0,C 180,E1 -10190.159,E2 -10190.159} C_VEL
LIN {X 0,Y 418.449,Z 203.116,A -85,B 0,C 180,E1 -10193.772,E2 -10193.772} C_VEL
LIN {X 0,Y 418.953,Z 194.498,A -85,B 0,C 180,E1 -10197.241,E2 -10197.241} C_VEL
LIN {X 0,Y 419.421,Z 187.495,A -85,B 0,C 180,E1 -10200.179,E2 -10200.179} C_VEL
LIN {X 0,Y 419.816,Z 182.373,A -85,B 0,C 180,E1 -10202.392,E2 -10202.392} C_VEL
LIN {X 0,Y 420.526,Z 174.969,A -85,B 0,C 180,E1 -10205.799,E2 -10205.799} C_VEL
LIN {X 0,Y 420.235,Z 171.419,A -85,B 0,C 180,E1 -10207.57,E2 -10207.57} C_VEL
LIN {X 0,Y 419.148,Z 165.122,A -85,B 0,C 180,E1 -10211.015,E2 -10211.015} C_VEL
LIN {X 0,Y 418.22,Z 160.391,A -85,B 0,C 180,E1 -10213.962,E2 -10213.962} C_VEL
LIN {X 0,Y 418.214,Z 160.396,A -85,B 0,C 180,E1 -10216.449,E2 -10216.449} C_VEL
LIN {X 0,Y 418.229,Z 160.394,A -85,B 0,C 180,E1 -10219.13,E2 -10219.13} C_VEL
LIN {X 0,Y 418.234,Z 160.391,A -85,B 0,C 180,E1 -10222.166,E2 -10222.166} C_VEL
LIN {X 0,Y 418.27,Z 160.385,A -85,B 0,C 180,E1 -10225.42,E2 -10225.42} C_VEL
LIN {X 0,Y 418.216,Z 160.392,A -85,B 0,C 180,E1 -10228.604,E2 -10228.604} C_VEL
LIN {X 0,Y 418.296,Z 160.382,A -85,B 0,C 180,E1 -10231.937,E2 -10231.937} C_VEL
LIN {X 0,Y 418.294,Z 160.381,A -85,B 0,C 180,E1 -10235.162,E2 -10235.162} C_VEL
LIN {X 0,Y 418.239,Z 160.389,A -85,B 0,C 180,E1 -10238.303,E2 -10238.303} C_VEL
LIN {X 0,Y 418.28,Z 160.384,A -85,B 0,C 180,E1 -10241.383,E2 -10241.383} C_VEL
LIN {X 0,Y 418.307,Z 160.381,A -85,B 0,C 180,E1 -10244.406,E2 -10244.406} C_VEL
LIN {X 0,Y 418.36,Z 160.374,A -85,B 0,C 180,E1 -10247.385,E2 -10247.385} C_VEL
LIN {X 0,Y 418.346,Z 160.377,A -85,B 0,C 180,E1 -10250.328,E2 -10250.328} C_VEL
LIN {X 0,Y 418.498,Z 160.357,A -85,B 0,C 180,E1 -10253.249,E2 -10253.249} C_VEL
LIN {X 0,Y 418.344,Z 160.376,A -85,B 0,C 180,E1 -10255.181,E2 -10255.181} C_VEL
LIN {X 0,Y 418.55,Z 160.351,A -85,B 0,C 180,E1 -10258.075,E2 -10258.075} C_VEL
LIN {X 0,Y 418.677,Z 160.335,A -85,B 0,C 180,E1 -10260,E2 -10260} C_VEL
LIN {X 0,Y 418.513,Z 160.356,A -85,B 0,C 180,E1 -10262.887,E2 -10262.887} C_VEL
LIN {X 0,Y 418.494,Z 160.361,A -85,B 0,C 180,E1 -10266.75,E2 -10266.75} C_VEL
LIN {X 0,Y 418.252,Z 160.389,A -85,B 0,C 180,E1 -10269.673,E2 -10269.673} C_VEL
LIN {X 0,Y 418.133,Z 160.406,A -85,B 0,C 180,E1 -10270.654,E2 -10270.654} C_VEL
LIN {X 0,Y 418.109,Z 162.156,A -85,B 0,C 180,E1 -10272.857,E2 -10272.857} C_VEL
LIN {X 0,Y 417.932,Z 165.733,A -85,B 0,C 180,E1 -10276.611,E2 -10276.611} C_VEL
LIN {X 0,Y 417.784,Z 168.681,A -85,B 0,C 180,E1 -10279.66,E2 -10279.66} C_VEL
LIN {X 0,Y 417.66,Z 171.716,A -85,B 0,C 180,E1 -10282.769,E2 -10282.769} C_VEL
LIN {X 0,Y 417.577,Z 174.864,A -85,B 0,C 180,E1 -10285.95,E2 -10285.95} C_VEL
LIN {X 0,Y 417.554,Z 176.757,A -85,B 0,C 180,E1 -10287.81,E2 -10287.81} C_VEL
LIN {X 0,Y 421.084,Z 189.9,A -85,B 0,C 180,E1 -10288.436,E2 -10288.436} C_VEL
LIN {X 0,Y 422.558,Z 196.951,A -85,B 0,C 180,E1 -10288.837,E2 -10288.837} C_VEL
LIN {X 0,Y 421.975,Z 208.88,A -85,B 0,C 180,E1 -10289.537,E2 -10289.537} C_VEL
LIN {X 0,Y 421.275,Z 220.713,A -85,B 0,C 180,E1 -10290.446,E2 -10290.446} C_VEL
LIN {X 0,Y 420.662,Z 231.052,A -85,B 0,C 180,E1 -10291.449,E2 -10291.449} C_VEL
LIN {X 0,Y 419.936,Z 240.936,A -85,B 0,C 180,E1 -10292.637,E2 -10292.637} C_VEL
LIN {X 0,Y 419.34,Z 249.128,A -85,B 0,C 180,E1 -10293.846,E2 -10293.846} C_VEL
LIN {X 0,Y 418.709,Z 256.122,A -85,B 0,C 180,E1 -10295.091,E2 -10295.091} C_VEL
LIN {X 0,Y 418.209,Z 263.398,A -85,B 0,C 180,E1 -10296.705,E2 -10296.705} C_VEL
LIN {X 0,Y 417.765,Z 269.531,A -85,B 0,C 180,E1 -10298.494,E2 -10298.494} C_VEL
LIN {X 0,Y 417.508,Z 272.865,A -85,B 0,C 180,E1 -10299.766,E2 -10299.766} C_VEL
LIN {X 0,Y 417.32,Z 275.415,A -85,B 0,C 180,E1 -10301.055,E2 -10301.055} C_VEL
LIN {X 0,Y 417.148,Z 277.218,A -85,B 0,C 180,E1 -10302.369,E2 -10302.369} C_VEL
LIN {X 0,Y 417.083,Z 278.287,A -85,B 0,C 180,E1 -10303.698,E2 -10303.698} C_VEL
LIN {X 0,Y 417.02,Z 278.615,A -85,B 0,C 180,E1 -10305.057,E2 -10305.057} C_VEL
LIN {X 0,Y 417.06,Z 278.113,A -85,B 0,C 180,E1 -10306.435,E2 -10306.435} C_VEL
LIN {X 0,Y 417.148,Z 276.756,A -85,B 0,C 180,E1 -10307.841,E2 -10307.841} C_VEL
LIN {X 0,Y 417.345,Z 274.489,A -85,B 0,C 180,E1 -10309.269,E2 -10309.269} C_VEL
LIN {X 0,Y 417.522,Z 271.165,A -85,B 0,C 180,E1 -10310.741,E2 -10310.741} C_VEL
LIN {X 0,Y 417.839,Z 266.659,A -85,B 0,C 180,E1 -10312.235,E2 -10312.235} C_VEL
LIN {X 0,Y 418.214,Z 260.728,A -85,B 0,C 180,E1 -10313.767,E2 -10313.767} C_VEL
LIN {X 0,Y 418.709,Z 253.012,A -85,B 0,C 180,E1 -10315.331,E2 -10315.331} C_VEL
LIN {X 0,Y 419.388,Z 244.592,A -85,B 0,C 180,E1 -10316.696,E2 -10316.696} C_VEL
LIN {X 0,Y 420.013,Z 234.828,A -85,B 0,C 180,E1 -10317.984,E2 -10317.984} C_VEL
LIN {X 0,Y 420.645,Z 224.394,A -85,B 0,C 180,E1 -10319.085,E2 -10319.085} C_VEL
LIN {X 0,Y 421.33,Z 212.287,A -85,B 0,C 180,E1 -10320.103,E2 -10320.103} C_VEL
LIN {X 0,Y 421.947,Z 201.109,A -85,B 0,C 180,E1 -10320.83,E2 -10320.83} C_VEL
LIN {X 0,Y 422.148,Z 195.459,A -85,B 0,C 180,E1 -10321.131,E2 -10321.131} C_VEL
LIN {X 0,Y 419.054,Z 181.848,A -85,B 0,C 180,E1 -10321.833,E2 -10321.833} C_VEL
LIN {X 0,Y 417.402,Z 175.104,A -85,B 0,C 180,E1 -10322.11,E2 -10322.11} C_VEL
LIN {X 0,Y 417.468,Z 171.581,A -85,B 0,C 180,E1 -10325.377,E2 -10325.377} C_VEL
LIN {X 0,Y 417.465,Z 168.521,A -85,B 0,C 180,E1 -10328.261,E2 -10328.261} C_VEL
LIN {X 0,Y 417.563,Z 165.306,A -85,B 0,C 180,E1 -10331.35,E2 -10331.35} C_VEL
LIN {X 0,Y 417.672,Z 162.17,A -85,B 0,C 180,E1 -10334.382,E2 -10334.382} C_VEL
LIN {X 0,Y 417.76,Z 160.452,A -85,B 0,C 180,E1 -10336.377,E2 -10336.377} C_VEL
LIN {X 0,Y 418.156,Z 160.397,A -85,B 0,C 180,E1 -10339.346,E2 -10339.346} C_VEL
LIN {X 0,Y 418.462,Z 160.362,A -85,B 0,C 180,E1 -10342.278,E2 -10342.278} C_VEL
LIN {X 0,Y 418.5,Z 160.357,A -85,B 0,C 180,E1 -10344.217,E2 -10344.217} C_VEL
LIN {X 0,Y 418.542,Z 160.352,A -85,B 0,C 180,E1 -10348.075,E2 -10348.075} C_VEL
LIN {X 0,Y 418.522,Z 160.351,A -85,B 0,C 180,E1 -10349.224,E2 -10349.224} C_VEL
LIN {X 0,Y 417.948,Z 160.427,A -85,B 0,C 180,E1 -10350.028,E2 -10350.028} C_VEL
LIN {X 0,Y 415.128,Z 160.775,A -85,B 0,C 180,E1 -10351.334,E2 -10351.334} C_VEL
LIN {X 0,Y 412.626,Z 161.087,A -85,B 0,C 180,E1 -10352.388,E2 -10352.388} C_VEL
LIN {X 0,Y 411.464,Z 161.23,A -85,B 0,C 180,E1 -10353.203,E2 -10353.203} C_VEL
LIN {X 0,Y 411.325,Z 161.247,A -85,B 0,C 180,E1 -10353.48,E2 -10353.48} C_VEL
LIN {X 0,Y 411.469,Z 161.234,A -85,B 0,C 180,E1 -10355.882,E2 -10355.882} C_VEL
LIN {X 0,Y 411.479,Z 161.232,A -85,B 0,C 180,E1 -10357.853,E2 -10357.853} C_VEL
LIN {X 0,Y 411.281,Z 161.257,A -85,B 0,C 180,E1 -10361.833,E2 -10361.833} C_VEL
LIN {X 0,Y 411.257,Z 161.256,A -85,B 0,C 180,E1 -10364.853,E2 -10364.853} C_VEL
LIN {X 0,Y 411.249,Z 161.26,A -85,B 0,C 180,E1 -10367.915,E2 -10367.915} C_VEL
LIN {X 0,Y 411.193,Z 161.266,A -85,B 0,C 180,E1 -10371.034,E2 -10371.034} C_VEL
LIN {X 0,Y 411.224,Z 161.26,A -85,B 0,C 180,E1 -10374.215,E2 -10374.215} C_VEL
LIN {X 0,Y 411.256,Z 161.26,A -85,B 0,C 180,E1 -10377.478,E2 -10377.478} C_VEL
LIN {X 0,Y 411.186,Z 161.267,A -85,B 0,C 180,E1 -10380.848,E2 -10380.848} C_VEL
LIN {X 0,Y 411.202,Z 161.262,A -85,B 0,C 180,E1 -10384.334,E2 -10384.334} C_VEL
LIN {X 0,Y 411.192,Z 161.264,A -85,B 0,C 180,E1 -10387.974,E2 -10387.974} C_VEL
LIN {X 0,Y 411.179,Z 161.267,A -85,B 0,C 180,E1 -10390.504,E2 -10390.504} C_VEL
LIN {X 0,Y 411.174,Z 161.27,A -85,B 0,C 180,E1 -10393.133,E2 -10393.133} C_VEL
LIN {X 0,Y 411.166,Z 161.268,A -85,B 0,C 180,E1 -10395.881,E2 -10395.881} C_VEL
LIN {X 0,Y 411.162,Z 161.271,A -85,B 0,C 180,E1 -10398.772,E2 -10398.772} C_VEL
LIN {X 0,Y 411.208,Z 161.262,A -85,B 0,C 180,E1 -10401.831,E2 -10401.831} C_VEL
LIN {X 0,Y 411.209,Z 161.265,A -85,B 0,C 180,E1 -10405.122,E2 -10405.122} C_VEL
LIN {X 0,Y 411.164,Z 161.268,A -85,B 0,C 180,E1 -10408.003,E2 -10408.003} C_VEL
LIN {X 0,Y 411.217,Z 161.262,A -85,B 0,C 180,E1 -10411.411,E2 -10411.411} C_VEL
LIN {X 0,Y 411.237,Z 161.258,A -85,B 0,C 180,E1 -10413.62,E2 -10413.62} C_VEL
LIN {X 0,Y 411.203,Z 161.265,A -85,B 0,C 180,E1 -10416.853,E2 -10416.853} C_VEL
LIN {X 0,Y 411.214,Z 161.263,A -85,B 0,C 180,E1 -10420.051,E2 -10420.051} C_VEL
LIN {X 0,Y 411.263,Z 161.256,A -85,B 0,C 180,E1 -10423.132,E2 -10423.132} C_VEL
LIN {X 0,Y 411.306,Z 161.252,A -85,B 0,C 180,E1 -10426.896,E2 -10426.896} C_VEL
LIN {X 0,Y 411.293,Z 161.255,A -85,B 0,C 180,E1 -10430.162,E2 -10430.162} C_VEL
LIN {X 0,Y 411.444,Z 161.233,A -85,B 0,C 180,E1 -10433.133,E2 -10433.133} C_VEL
LIN {X 0,Y 411.312,Z 161.248,A -85,B 0,C 180,E1 -10435.1,E2 -10435.1} C_VEL
LIN {X 0,Y 411.515,Z 161.228,A -85,B 0,C 180,E1 -10438.043,E2 -10438.043} C_VEL
LIN {X 0,Y 411.642,Z 161.211,A -85,B 0,C 180,E1 -10440.001,E2 -10440.001} C_VEL
LIN {X 0,Y 411.459,Z 161.231,A -85,B 0,C 180,E1 -10442.938,E2 -10442.938} C_VEL
LIN {X 0,Y 411.426,Z 161.235,A -85,B 0,C 180,E1 -10446.868,E2 -10446.868} C_VEL
LIN {X 0,Y 411.293,Z 161.255,A -85,B 0,C 180,E1 -10449.839,E2 -10449.839} C_VEL
LIN {X 0,Y 411.307,Z 161.251,A -85,B 0,C 180,E1 -10453.105,E2 -10453.105} C_VEL
LIN {X 0,Y 411.259,Z 161.256,A -85,B 0,C 180,E1 -10456.889,E2 -10456.889} C_VEL
LIN {X 0,Y 411.233,Z 161.261,A -85,B 0,C 180,E1 -10459.987,E2 -10459.987} C_VEL
LIN {X 0,Y 411.206,Z 161.264,A -85,B 0,C 180,E1 -10463.148,E2 -10463.148} C_VEL
LIN {X 0,Y 411.24,Z 161.257,A -85,B 0,C 180,E1 -10466.381,E2 -10466.381} C_VEL
LIN {X 0,Y 411.203,Z 161.265,A -85,B 0,C 180,E1 -10469.713,E2 -10469.713} C_VEL
LIN {X 0,Y 411.208,Z 161.266,A -85,B 0,C 180,E1 -10473.156,E2 -10473.156} C_VEL
LIN {X 0,Y 411.194,Z 161.264,A -85,B 0,C 180,E1 -10476.553,E2 -10476.553} C_VEL
LIN {X 0,Y 411.213,Z 161.263,A -85,B 0,C 180,E1 -10479.728,E2 -10479.728} C_VEL
LIN {X 0,Y 411.176,Z 161.264,A -85,B 0,C 180,E1 -10483.134,E2 -10483.134} C_VEL
LIN {X 0,Y 411.175,Z 161.333,A -85,B 0,C 180,E1 -10486.401,E2 -10486.401} C_VEL
LIN {X 0,Y 412.338,Z 167.354,A -85,B 0,C 180,E1 -10489.633,E2 -10489.633} C_VEL
LIN {X 0,Y 413.232,Z 172.519,A -85,B 0,C 180,E1 -10492.246,E2 -10492.246} C_VEL
LIN {X 0,Y 413.529,Z 176.369,A -85,B 0,C 180,E1 -10494.103,E2 -10494.103} C_VEL
LIN {X 0,Y 412.964,Z 184.109,A -85,B 0,C 180,E1 -10497.583,E2 -10497.583} C_VEL
LIN {X 0,Y 412.304,Z 191.881,A -85,B 0,C 180,E1 -10500.935,E2 -10500.935} C_VEL
LIN {X 0,Y 411.806,Z 199.684,A -85,B 0,C 180,E1 -10504.203,E2 -10504.203} C_VEL
LIN {X 0,Y 411.26,Z 208.867,A -85,B 0,C 180,E1 -10507.917,E2 -10507.917} C_VEL
LIN {X 0,Y 410.893,Z 216.714,A -85,B 0,C 180,E1 -10511.036,E2 -10511.036} C_VEL
LIN {X 0,Y 410.729,Z 220.192,A -85,B 0,C 180,E1 -10512.393,E2 -10512.393} C_VEL
LIN {X 0,Y 413.111,Z 235.056,A -85,B 0,C 180,E1 -10512.969,E2 -10512.969} C_VEL
LIN {X 0,Y 414.844,Z 247.629,A -85,B 0,C 180,E1 -10513.641,E2 -10513.641} C_VEL
LIN {X 0,Y 414.26,Z 259.339,A -85,B 0,C 180,E1 -10514.376,E2 -10514.376} C_VEL
LIN {X 0,Y 413.544,Z 270.047,A -85,B 0,C 180,E1 -10515.231,E2 -10515.231} C_VEL
LIN {X 0,Y 412.87,Z 279.941,A -85,B 0,C 180,E1 -10516.213,E2 -10516.213} C_VEL
LIN {X 0,Y 412.156,Z 289.964,A -85,B 0,C 180,E1 -10517.443,E2 -10517.443} C_VEL
LIN {X 0,Y 411.444,Z 298.187,A -85,B 0,C 180,E1 -10518.672,E2 -10518.672} C_VEL
LIN {X 0,Y 410.898,Z 306.268,A -85,B 0,C 180,E1 -10520.152,E2 -10520.152} C_VEL
LIN {X 0,Y 410.483,Z 312.76,A -85,B 0,C 180,E1 -10521.632,E2 -10521.632} C_VEL
LIN {X 0,Y 410.195,Z 317.915,A -85,B 0,C 180,E1 -10523.112,E2 -10523.112} C_VEL
LIN {X 0,Y 410.1,Z 321.921,A -85,B 0,C 180,E1 -10524.592,E2 -10524.592} C_VEL
LIN {X 0,Y 409.953,Z 324.87,A -85,B 0,C 180,E1 -10526.068,E2 -10526.068} C_VEL
LIN {X 0,Y 409.993,Z 326.28,A -85,B 0,C 180,E1 -10527.052,E2 -10527.052} C_VEL
LIN {X 0,Y 409.989,Z 327.279,A -85,B 0,C 180,E1 -10528.035,E2 -10528.035} C_VEL
LIN {X 0,Y 409.956,Z 328.091,A -85,B 0,C 180,E1 -10530,E2 -10530} C_VEL
LIN {X 0,Y 409.948,Z 327.86,A -85,B 0,C 180,E1 -10530.982,E2 -10530.982} C_VEL
LIN {X 0,Y 409.989,Z 327.233,A -85,B 0,C 180,E1 -10531.965,E2 -10531.965} C_VEL
LIN {X 0,Y 410.007,Z 326.211,A -85,B 0,C 180,E1 -10532.948,E2 -10532.948} C_VEL
LIN {X 0,Y 409.955,Z 324.777,A -85,B 0,C 180,E1 -10533.932,E2 -10533.932} C_VEL
LIN {X 0,Y 410.109,Z 321.787,A -85,B 0,C 180,E1 -10535.409,E2 -10535.409} C_VEL
LIN {X 0,Y 410.199,Z 317.738,A -85,B 0,C 180,E1 -10536.888,E2 -10536.888} C_VEL
